(* IEC 61131-3 sources: SmartHomeNew/snapshots/2026-05-25 (part 5) *)

(* ---- PRG_Forensic_Evidence_Governor.st ---- *)
PROGRAM PRG_Forensic_Evidence_Governor
VAR
    L_Now_MS : UDINT;
    L_Forensic_Valid : BOOL := TRUE;
    L_Error_Code : UDINT := 0;
    L_Error_Text : STRING(160) := '';
END_VAR

L_Now_MS := GVL_STATUS.G_System_Time_MS;
L_Forensic_Valid := TRUE;
L_Error_Code := 0;
L_Error_Text := '';

// Fail-safe defaults.
GVL_FORENSIC_EVIDENCE_FABRIC.Forensic_Evidence_Valid := FALSE;
GVL_FORENSIC_EVIDENCE_FABRIC.Forensic_Evidence_Granted := FALSE;
GVL_FORENSIC_EVIDENCE_FABRIC.Forensic_Evidence_Quarantine_Active := TRUE;

GVL_FORENSIC_EVIDENCE_FABRIC.Authority_Lineage_Reconstructable := FALSE;
GVL_FORENSIC_EVIDENCE_FABRIC.Decision_Causality_Traceable := FALSE;
GVL_FORENSIC_EVIDENCE_FABRIC.Distributed_Evidence_Coherent := FALSE;
GVL_FORENSIC_EVIDENCE_FABRIC.Immutable_Audit_Continuity_Valid := FALSE;
GVL_FORENSIC_EVIDENCE_FABRIC.Recovery_Lineage_Preserved := FALSE;

// Compliance federation required.
IF NOT GVL_COMPLIANCE_FEDERATION_FABRIC.Compliance_Federation_Granted THEN
    L_Forensic_Valid := FALSE;
    L_Error_Code := 43000;
    L_Error_Text := 'Compliance federation authority not granted';
END_IF;

// Forensic split-brain detectors.
IF GVL_FORENSIC_EVIDENCE_FABRIC.Authority_Lineage_Gap_Detected THEN
    L_Forensic_Valid := FALSE;
    L_Error_Code := 43001;
    L_Error_Text := 'Authority lineage gap detected';
END_IF;

IF GVL_FORENSIC_EVIDENCE_FABRIC.NonReconstructable_Decision_Detected THEN
    L_Forensic_Valid := FALSE;
    L_Error_Code := 43002;
    L_Error_Text := 'Non-reconstructable decision detected';
END_IF;

IF GVL_FORENSIC_EVIDENCE_FABRIC.History_Evidence_Divergence_Detected THEN
    L_Forensic_Valid := FALSE;
    L_Error_Code := 43003;
    L_Error_Text := 'History evidence divergence detected';
END_IF;

IF GVL_FORENSIC_EVIDENCE_FABRIC.Causal_Chain_Erosion_Detected THEN
    L_Forensic_Valid := FALSE;
    L_Error_Code := 43004;
    L_Error_Text := 'Causal chain erosion detected';
END_IF;

IF GVL_FORENSIC_EVIDENCE_FABRIC.Distributed_Forensic_Inconsistency_Detected THEN
    L_Forensic_Valid := FALSE;
    L_Error_Code := 43005;
    L_Error_Text := 'Distributed forensic inconsistency detected';
END_IF;

IF GVL_FORENSIC_EVIDENCE_FABRIC.Immutable_Audit_Discontinuity_Detected THEN
    L_Forensic_Valid := FALSE;
    L_Error_Code := 43006;
    L_Error_Text := 'Immutable audit discontinuity detected';
END_IF;

// Forensic reconstruction validation.
IF L_Forensic_Valid
AND NOT GVL_FORENSIC_EVIDENCE_FABRIC.Historical_Proof_Chain_Valid THEN
    L_Forensic_Valid := FALSE;
    L_Error_Code := 43010;
    L_Error_Text := 'Historical proof chain invalid';
END_IF;

IF L_Forensic_Valid
AND NOT GVL_FORENSIC_EVIDENCE_FABRIC.Governance_Event_Lineage_Coherent THEN
    L_Forensic_Valid := FALSE;
    L_Error_Code := 43011;
    L_Error_Text := 'Governance event lineage coherence invalid';
END_IF;

IF L_Forensic_Valid
AND NOT GVL_FORENSIC_EVIDENCE_FABRIC.Semantic_Transition_Traceable THEN
    L_Forensic_Valid := FALSE;
    L_Error_Code := 43012;
    L_Error_Text := 'Semantic transition traceability invalid';
END_IF;

IF L_Forensic_Valid
AND NOT GVL_FORENSIC_EVIDENCE_FABRIC.Physical_Transition_Traceable THEN
    L_Forensic_Valid := FALSE;
    L_Error_Code := 43013;
    L_Error_Text := 'Physical transition traceability invalid';
END_IF;

IF L_Forensic_Valid THEN
    GVL_FORENSIC_EVIDENCE_FABRIC.Forensic_Evidence_Valid := TRUE;
    GVL_FORENSIC_EVIDENCE_FABRIC.Forensic_Evidence_Granted := TRUE;
    GVL_FORENSIC_EVIDENCE_FABRIC.Forensic_Evidence_Quarantine_Active := FALSE;

    GVL_FORENSIC_EVIDENCE_FABRIC.Authority_Lineage_Reconstructable := TRUE;
    GVL_FORENSIC_EVIDENCE_FABRIC.Decision_Causality_Traceable := TRUE;
    GVL_FORENSIC_EVIDENCE_FABRIC.Distributed_Evidence_Coherent := TRUE;
    GVL_FORENSIC_EVIDENCE_FABRIC.Immutable_Audit_Continuity_Valid := TRUE;
    GVL_FORENSIC_EVIDENCE_FABRIC.Recovery_Lineage_Preserved := TRUE;

    GVL_FORENSIC_EVIDENCE_FABRIC.Forensic_Evidence_Epoch :=
        GVL_COMPLIANCE_FEDERATION_FABRIC.Compliance_Federation_Epoch;

    GVL_FORENSIC_EVIDENCE_FABRIC.Forensic_Evidence_Epoch_Coherent := TRUE;

    GVL_FORENSIC_EVIDENCE_FABRIC.Forensic_Evidence_Last_Update_MS :=
        L_Now_MS;

    GVL_FORENSIC_EVIDENCE_FABRIC.Forensic_Evidence_Lease_Expired := FALSE;

    GVL_FORENSIC_EVIDENCE_FABRIC.Forensic_Evidence_Last_Error_Code := 0;
    GVL_FORENSIC_EVIDENCE_FABRIC.Forensic_Evidence_Last_Error_Text := '';
ELSE
    GVL_FORENSIC_EVIDENCE_FABRIC.Forensic_Evidence_Valid := FALSE;
    GVL_FORENSIC_EVIDENCE_FABRIC.Forensic_Evidence_Granted := FALSE;
    GVL_FORENSIC_EVIDENCE_FABRIC.Forensic_Evidence_Quarantine_Active := TRUE;

    GVL_FORENSIC_EVIDENCE_FABRIC.Forensic_Evidence_Lease_Expired := TRUE;

    GVL_FORENSIC_EVIDENCE_FABRIC.Forensic_Evidence_Last_Error_Code :=
        L_Error_Code;

    GVL_FORENSIC_EVIDENCE_FABRIC.Forensic_Evidence_Last_Error_Text :=
        L_Error_Text;

    GVL_FORENSIC_EVIDENCE_FABRIC.Forensic_Evidence_Invalidation_Count :=
        GVL_FORENSIC_EVIDENCE_FABRIC.Forensic_Evidence_Invalidation_Count + 1;
END_IF;

END_PROGRAM

(* ---- PRG_Governance_Liveness_Integrity_Governor.st ---- *)
PROGRAM PRG_Governance_Liveness_Integrity_Governor
VAR
    L_Now_MS : UDINT;
    L_Integrity_Valid : BOOL := TRUE;
    L_Error_Code : UDINT := 0;
    L_Error_Text : STRING(160) := '';
END_VAR

L_Now_MS := GVL_STATUS.G_System_Time_MS;
L_Integrity_Valid := TRUE;
L_Error_Code := 0;
L_Error_Text := '';

// Fail-safe defaults.
GVL_GOVERNANCE_LIVENESS_INTEGRITY_FABRIC.Governance_Liveness_Integrity_Valid := FALSE;
GVL_GOVERNANCE_LIVENESS_INTEGRITY_FABRIC.Governance_Liveness_Integrity_Granted := FALSE;
GVL_GOVERNANCE_LIVENESS_INTEGRITY_FABRIC.Governance_Liveness_Integrity_Quarantine_Active := TRUE;

GVL_GOVERNANCE_LIVENESS_INTEGRITY_FABRIC.Governance_Execution_Liveness_Stable := FALSE;
GVL_GOVERNANCE_LIVENESS_INTEGRITY_FABRIC.Integrity_Governor_Scheduling_Canonical := FALSE;
GVL_GOVERNANCE_LIVENESS_INTEGRITY_FABRIC.CrossGovernor_Execution_Continuity_Valid := FALSE;
GVL_GOVERNANCE_LIVENESS_INTEGRITY_FABRIC.Deterministic_Validation_Cycle_Integrity := FALSE;
GVL_GOVERNANCE_LIVENESS_INTEGRITY_FABRIC.Governance_Runtime_Liveness_Coherent := FALSE;

// Governance validator integrity required.
IF NOT GVL_GOVERNANCE_VALIDATOR_INTEGRITY_FABRIC.Governance_Validator_Integrity_Granted THEN
    L_Integrity_Valid := FALSE;
    L_Error_Code := 54000;
    L_Error_Text := 'Governance validator integrity not granted';
END_IF;

// Governance liveness degradation detectors.
IF GVL_GOVERNANCE_LIVENESS_INTEGRITY_FABRIC.Integrity_Governor_Starvation_Detected THEN
    L_Integrity_Valid := FALSE;
    L_Error_Code := 54001;
    L_Error_Text := 'Integrity governor starvation detected';
END_IF;

IF GVL_GOVERNANCE_LIVENESS_INTEGRITY_FABRIC.Validation_Cycle_Skip_Detected THEN
    L_Integrity_Valid := FALSE;
    L_Error_Code := 54002;
    L_Error_Text := 'Validation cycle skip detected';
END_IF;

IF GVL_GOVERNANCE_LIVENESS_INTEGRITY_FABRIC.CrossGovernor_Execution_Jitter_Fork THEN
    L_Integrity_Valid := FALSE;
    L_Error_Code := 54003;
    L_Error_Text := 'Cross-governor execution jitter fork detected';
END_IF;

IF GVL_GOVERNANCE_LIVENESS_INTEGRITY_FABRIC.Selective_Governance_Degradation_Detected THEN
    L_Integrity_Valid := FALSE;
    L_Error_Code := 54004;
    L_Error_Text := 'Selective governance degradation detected';
END_IF;

IF GVL_GOVERNANCE_LIVENESS_INTEGRITY_FABRIC.Runtime_Governor_Execution_Stall_Detected THEN
    L_Integrity_Valid := FALSE;
    L_Error_Code := 54005;
    L_Error_Text := 'Runtime governor execution stall detected';
END_IF;

IF GVL_GOVERNANCE_LIVENESS_INTEGRITY_FABRIC.Distributed_Liveness_Reality_Fork_Detected THEN
    L_Integrity_Valid := FALSE;
    L_Error_Code := 54006;
    L_Error_Text := 'Distributed liveness reality fork detected';
END_IF;

// Governance liveness validation.
IF L_Integrity_Valid
AND NOT GVL_GOVERNANCE_LIVENESS_INTEGRITY_FABRIC.Validation_Cycle_Timing_Monotonic THEN
    L_Integrity_Valid := FALSE;
    L_Error_Code := 54010;
    L_Error_Text := 'Validation cycle timing invalid';
END_IF;

IF L_Integrity_Valid
AND NOT GVL_GOVERNANCE_LIVENESS_INTEGRITY_FABRIC.Distributed_Governor_Execution_Aligned THEN
    L_Integrity_Valid := FALSE;
    L_Error_Code := 54011;
    L_Error_Text := 'Distributed governor execution alignment invalid';
END_IF;

IF L_Integrity_Valid
AND NOT GVL_GOVERNANCE_LIVENESS_INTEGRITY_FABRIC.Runtime_Integrity_Causality_Grounded THEN
    L_Integrity_Valid := FALSE;
    L_Error_Code := 54012;
    L_Error_Text := 'Runtime integrity causality invalid';
END_IF;

IF L_Integrity_Valid
AND NOT GVL_GOVERNANCE_LIVENESS_INTEGRITY_FABRIC.Governance_Execution_Budget_Stable THEN
    L_Integrity_Valid := FALSE;
    L_Error_Code := 54013;
    L_Error_Text := 'Governance execution budget invalid';
END_IF;

IF L_Integrity_Valid THEN
    GVL_GOVERNANCE_LIVENESS_INTEGRITY_FABRIC.Governance_Liveness_Integrity_Valid := TRUE;
    GVL_GOVERNANCE_LIVENESS_INTEGRITY_FABRIC.Governance_Liveness_Integrity_Granted := TRUE;
    GVL_GOVERNANCE_LIVENESS_INTEGRITY_FABRIC.Governance_Liveness_Integrity_Quarantine_Active := FALSE;

    GVL_GOVERNANCE_LIVENESS_INTEGRITY_FABRIC.Governance_Execution_Liveness_Stable := TRUE;
    GVL_GOVERNANCE_LIVENESS_INTEGRITY_FABRIC.Integrity_Governor_Scheduling_Canonical := TRUE;
    GVL_GOVERNANCE_LIVENESS_INTEGRITY_FABRIC.CrossGovernor_Execution_Continuity_Valid := TRUE;
    GVL_GOVERNANCE_LIVENESS_INTEGRITY_FABRIC.Deterministic_Validation_Cycle_Integrity := TRUE;
    GVL_GOVERNANCE_LIVENESS_INTEGRITY_FABRIC.Governance_Runtime_Liveness_Coherent := TRUE;

    GVL_GOVERNANCE_LIVENESS_INTEGRITY_FABRIC.Governance_Liveness_Integrity_Epoch :=
        GVL_GOVERNANCE_VALIDATOR_INTEGRITY_FABRIC.Governance_Validator_Integrity_Epoch;

    GVL_GOVERNANCE_LIVENESS_INTEGRITY_FABRIC.Governance_Liveness_Integrity_Epoch_Coherent := TRUE;

    GVL_GOVERNANCE_LIVENESS_INTEGRITY_FABRIC.Governance_Liveness_Integrity_Last_Update_MS :=
        L_Now_MS;

    GVL_GOVERNANCE_LIVENESS_INTEGRITY_FABRIC.Governance_Liveness_Integrity_Lease_Expired := FALSE;

    GVL_GOVERNANCE_LIVENESS_INTEGRITY_FABRIC.Governance_Liveness_Integrity_Last_Error_Code := 0;
    GVL_GOVERNANCE_LIVENESS_INTEGRITY_FABRIC.Governance_Liveness_Integrity_Last_Error_Text := '';
ELSE
    GVL_GOVERNANCE_LIVENESS_INTEGRITY_FABRIC.Governance_Liveness_Integrity_Valid := FALSE;
    GVL_GOVERNANCE_LIVENESS_INTEGRITY_FABRIC.Governance_Liveness_Integrity_Granted := FALSE;
    GVL_GOVERNANCE_LIVENESS_INTEGRITY_FABRIC.Governance_Liveness_Integrity_Quarantine_Active := TRUE;

    GVL_GOVERNANCE_LIVENESS_INTEGRITY_FABRIC.Governance_Liveness_Integrity_Lease_Expired := TRUE;

    GVL_GOVERNANCE_LIVENESS_INTEGRITY_FABRIC.Governance_Liveness_Integrity_Last_Error_Code :=
        L_Error_Code;

    GVL_GOVERNANCE_LIVENESS_INTEGRITY_FABRIC.Governance_Liveness_Integrity_Last_Error_Text :=
        L_Error_Text;

    GVL_GOVERNANCE_LIVENESS_INTEGRITY_FABRIC.Governance_Liveness_Integrity_Invalidation_Count :=
        GVL_GOVERNANCE_LIVENESS_INTEGRITY_FABRIC.Governance_Liveness_Integrity_Invalidation_Count + 1;
END_IF;

END_PROGRAM

(* ---- PRG_HA_Session_Replication.st ---- *)
PROGRAM PRG_HA_Session_Replication
// ======================================================
// HA SESSION REPLICATION
// ======================================================
// Dedicated HA/session replication boundary.
//
// Purpose:
// replicate canonical peer-session state through isolated
// HA replication surface.
//
// Current implementation:
// bounded loopback foundation.
//
// Future implementations may replace this with:
// - SysCom HA channel
// - shared-memory replication
// - dedicated Ethernet HA link
// - deterministic fieldbus synchronization
//
// without changing distributed governors.
// ======================================================

IF NOT GVL_HA_SESSION_REPLICATION.HA_Replication_Enabled THEN
    GVL_HA_SESSION_REPLICATION.HA_Channel_Healthy := FALSE;
    RETURN;
END_IF;

// ------------------------------------------------------
// Canonical session export replication.
// ------------------------------------------------------

GVL_HA_SESSION_REPLICATION.HA_Remote_Session_Valid :=
    GVL_PEER_SESSION.Remote_Session_Valid;

GVL_HA_SESSION_REPLICATION.HA_Remote_Last_Refresh_MS :=
    GVL_PEER_SESSION.Remote_Last_Refresh_MS;

GVL_HA_SESSION_REPLICATION.HA_Remote_Runtime_Epoch :=
    GVL_PEER_SESSION.Remote_Runtime_Epoch;

GVL_HA_SESSION_REPLICATION.HA_Remote_Snapshot_Epoch :=
    GVL_PEER_SESSION.Remote_Snapshot_Epoch;

GVL_HA_SESSION_REPLICATION.HA_Remote_Boot_Generation :=
    GVL_PEER_SESSION.Remote_Boot_Generation;

GVL_HA_SESSION_REPLICATION.HA_Remote_Fencing_Token :=
    GVL_PEER_SESSION.Remote_Fencing_Token;

GVL_HA_SESSION_REPLICATION.HA_Remote_Publication_Allowed :=
    GVL_PEER_SESSION.Remote_Publication_Allowed;

GVL_HA_SESSION_REPLICATION.HA_Remote_Runtime_Healthy :=
    GVL_PEER_SESSION.Remote_Runtime_Healthy;

GVL_HA_SESSION_REPLICATION.HA_Last_TX_MS :=
    GVL_STATUS.G_System_Time_MS;

GVL_HA_SESSION_REPLICATION.HA_Last_RX_MS :=
    GVL_STATUS.G_System_Time_MS;

GVL_HA_SESSION_REPLICATION.HA_Channel_Healthy := TRUE;

// >>> BULK_SYNC_ANCHOR: PRG_HA_Session_Replication <<<
END_PROGRAM

(* ---- PRG_Heating_Config_Defaults.st ---- *)
PROGRAM PRG_Heating_Config_Defaults
VAR
    L_i : INT;
    L_Manifold : BYTE;
END_VAR

// Default per-circuit comfort/economy profiles.
// This initializer only fills empty records and does not overwrite HMI-edited
// records after circuit_id has been assigned.
FOR L_i := 1 TO GVL_CONSTANTS.C_MAX_HEATING_CIRCUITS DO
    IF GVL_CONFIG.G_HMI_FloorHeating_Configs[L_i].circuit_id = 0 THEN
        CASE L_i OF
            1, 2, 3, 4:
                L_Manifold := 1;
            5, 6, 7, 8:
                L_Manifold := 2;
            9, 10, 11, 12:
                L_Manifold := 3;
            13, 14:
                L_Manifold := 4;
        ELSE
                L_Manifold := 5;
        END_CASE;

        GVL_CONFIG.G_HMI_FloorHeating_Configs[L_i].circuit_id := TO_BYTE(L_i);
        GVL_CONFIG.G_HMI_FloorHeating_Configs[L_i].zone := TO_BYTE(L_i);
        GVL_CONFIG.G_HMI_FloorHeating_Configs[L_i].manifold_id := L_Manifold;
        GVL_CONFIG.G_HMI_FloorHeating_Configs[L_i].sensor_id := TO_BYTE(L_i);
        GVL_CONFIG.G_HMI_FloorHeating_Configs[L_i].valve_id := TO_BYTE(L_i);
        GVL_CONFIG.G_HMI_FloorHeating_Configs[L_i].control_type := 1;

        // Historical design_temp is kept, but explicit comfort_temp is now the
        // room comfort setpoint used by FB_Heating_Circuit_Control.
        GVL_CONFIG.G_HMI_FloorHeating_Configs[L_i].design_temp := 22.0;
        GVL_CONFIG.G_HMI_FloorHeating_Configs[L_i].use_in_normal := TRUE;
        GVL_CONFIG.G_HMI_FloorHeating_Configs[L_i].use_in_away_preheat := TRUE;
        GVL_CONFIG.G_HMI_FloorHeating_Configs[L_i].comfort_temp := 22.0;
        GVL_CONFIG.G_HMI_FloorHeating_Configs[L_i].economy_temp := 17.0;
        GVL_CONFIG.G_HMI_FloorHeating_Configs[L_i].long_away_temp := 12.0;

        GVL_CONFIG.G_HMI_FloorHeating_Configs[L_i].min_temp := 5.0;
        GVL_CONFIG.G_HMI_FloorHeating_Configs[L_i].max_temp := 30.0;
        GVL_CONFIG.G_HMI_FloorHeating_Configs[L_i].pid_kp := 2.0;
        GVL_CONFIG.G_HMI_FloorHeating_Configs[L_i].pwm_period_s := 600;
    END_IF;
END_FOR;

PRG_Away_Heating_HMI_Applicator();

END_PROGRAM

(* ---- PRG_Industrial_Maintainability_Governor.st ---- *)
PROGRAM PRG_Industrial_Maintainability_Governor

// Passive maintainability governance placeholder.
// Runtime maintainability state is currently represented by fabric GVLs only.
// This program is intentionally side-effect free until ownership is formalized.

END_PROGRAM

(* ---- PRG_Input_Quality_Read.st ---- *)
PROGRAM PRG_Input_Quality_Read
VAR
    L_i : INT;
    fbRoomTempQuality : ARRAY[1..GVL_CONSTANTS.C_MAX_ZONES] OF FB_Input_Quality_Observer;
    fbFloorTempQuality : ARRAY[1..GVL_CONSTANTS.C_MAX_HEATING_CIRCUITS] OF FB_Input_Quality_Observer;
END_VAR

FOR L_i := 1 TO GVL_CONSTANTS.C_MAX_ZONES DO
    fbRoomTempQuality[L_i](
        VI_Enable := GVL_INPUT_VALIDATION_CONFIG.G_Enable_Temporal_Anomaly_Detection,
        VI_Value := GVL_STATE.G_Room_Temps[L_i],
        VI_System_Time_MS := GVL_STATUS.G_System_Time_MS,
        VI_Spike_Threshold := GVL_INPUT_VALIDATION_CONFIG.G_Room_Temp_Spike_Threshold,
        VI_Stuck_Timeout_MS := GVL_INPUT_VALIDATION_CONFIG.G_Sensor_Stuck_Timeout_MS,
        VO_Quality => GVL_INPUT_QUALITY.G_Room_Temp_Quality[L_i]
    );
END_FOR;

FOR L_i := 1 TO GVL_CONSTANTS.C_MAX_HEATING_CIRCUITS DO
    fbFloorTempQuality[L_i](
        VI_Enable := GVL_INPUT_VALIDATION_CONFIG.G_Enable_Temporal_Anomaly_Detection,
        VI_Value := GVL_STATE.G_Floor_Temps[L_i],
        VI_System_Time_MS := GVL_STATUS.G_System_Time_MS,
        VI_Spike_Threshold := GVL_INPUT_VALIDATION_CONFIG.G_Room_Temp_Spike_Threshold,
        VI_Stuck_Timeout_MS := GVL_INPUT_VALIDATION_CONFIG.G_Sensor_Stuck_Timeout_MS,
        VO_Quality => GVL_INPUT_QUALITY.G_Floor_Temp_Quality[L_i]
    );
END_FOR;

END_PROGRAM

(* ---- PRG_IO_Read_Discrete_03_Safety_Sensors.st ---- *)
PROGRAM PRG_IO_Read_Discrete_03_Safety_Sensors
VAR
    L_i : INT;
    L_Debounce_Time : TIME := T#100MS;

    fbDebounce_Flood : ARRAY[1..GVL_CONSTANTS.C_MAX_FLOOD_SENSORS] OF FB_System_Timer;
    fbDebounce_Smoke : ARRAY[1..GVL_CONSTANTS.C_MAX_SMOKE_SENSORS] OF FB_System_Timer;
END_VAR

FOR L_i := 1 TO GVL_CONSTANTS.C_MAX_FLOOD_SENSORS DO
    fbDebounce_Flood[L_i](
        IN := GVL_IO.DI_Flood_Sensors[L_i],
        PT := L_Debounce_Time,
        VI_System_Time_MS := GVL_STATUS.G_System_Time_MS
    );
    GVL_STATE.G_Water_Sensors[L_i] := fbDebounce_Flood[L_i].Q;
END_FOR;

FOR L_i := 1 TO GVL_CONSTANTS.C_MAX_SMOKE_SENSORS DO
    fbDebounce_Smoke[L_i](
        IN := GVL_IO.DI_Smoke_Sensors[L_i],
        PT := L_Debounce_Time,
        VI_System_Time_MS := GVL_STATUS.G_System_Time_MS
    );
    GVL_STATE.G_Smoke_Sensors[L_i] := fbDebounce_Smoke[L_i].Q;
END_FOR;

// >>> BULK_SYNC_ANCHOR: PRG_IO_Read_Discrete_03_Safety_Sensors <<<
END_PROGRAM

(* ---- PRG_IO_Read_Manifold_01_Pressure_Current.st ---- *)
PROGRAM PRG_IO_Read_Manifold_01_Pressure_Current
VAR
    L_i : INT;
    L_Manifold_Pressure_Raw : WORD;
    L_Manifold_Current_Raw : WORD;

    fbDiagEventManager : FB_Diagnostics_Event_Manager;
    fbAnalog_Manifold_Pressure : ARRAY[1..GVL_CONSTANTS.C_MAX_MANIFOLDS] OF FB_Sensor_Analog_Processing;
    fbAnalog_Manifold_Current : ARRAY[1..GVL_CONSTANTS.C_MAX_MANIFOLDS] OF FB_Sensor_Analog_Processing;
END_VAR

GVL_STATUS.G_Diagnostics.Manifold_Pressure_Fault_Active := FALSE;
GVL_STATUS.G_Diagnostics.Manifold_Pressure_First_Fault_Index := 0;
GVL_STATUS.G_Diagnostics.Manifold_Current_Fault_Active := FALSE;
GVL_STATUS.G_Diagnostics.Manifold_Current_First_Fault_Index := 0;
GVL_STATUS.G_Diagnostics.Manifold_Pressure_Fault_Text := '';
GVL_STATUS.G_Diagnostics.Manifold_Current_Fault_Text := '';

FOR L_i := 1 TO GVL_CONSTANTS.C_MAX_MANIFOLDS DO
    IF GVL_IO.AI_Manifold_Pressures[L_i] < 0 THEN
        L_Manifold_Pressure_Raw := 0;
    ELSE
        L_Manifold_Pressure_Raw := INT_TO_WORD(GVL_IO.AI_Manifold_Pressures[L_i]);
    END_IF;

    IF GVL_IO.AI_Manifold_Currents[L_i] < 0 THEN
        L_Manifold_Current_Raw := 0;
    ELSE
        L_Manifold_Current_Raw := INT_TO_WORD(GVL_IO.AI_Manifold_Currents[L_i]);
    END_IF;

    fbAnalog_Manifold_Pressure[L_i](
        VI_Raw_Value := L_Manifold_Pressure_Raw,
        VI_Sensor_Type := 0,
        VI_Min_Scale := 0.0,
        VI_Max_Scale := 10.0,
        VI_Offset := 0.0,
        VI_Multiplier := 1.0,
        VI_Filter_Time_MS := GVL_CONSTANTS.C_MS_IN_SECOND,
        VI_System_Time_MS := GVL_STATUS.G_System_Time_MS,
        VI_Fallback_Mode := 0,
        VI_Default_Value := 0.0
    );
    GVL_STATE.G_Manifold_Pressures[L_i] := fbAnalog_Manifold_Pressure[L_i].VO_Value;
    GVL_STATUS.G_Diagnostics.Manifold_Pressure_Fault[L_i] := fbAnalog_Manifold_Pressure[L_i].VO_Error;
    GVL_STATUS.G_Diagnostics.Manifold_Pressure_Diag_Code[L_i] := fbAnalog_Manifold_Pressure[L_i].VO_Diag_Code;

    fbDiagEventManager(
        VI_Code := GVL_CONFIG.ERR_PRESSURE_OUT_OF_RANGE,
        VI_Severity := 3,
        VI_Active := fbAnalog_Manifold_Pressure[L_i].VO_Error,
        VI_Timestamp := GVL_STATUS.G_System_Time_MS,
        VI_Source := 100 + L_i,
        VIO_Events := GVL_STATUS.G_Diagnostics_Events,
        VIO_Count := GVL_STATUS.G_Diagnostics_Count
    );

    fbAnalog_Manifold_Current[L_i](
        VI_Raw_Value := L_Manifold_Current_Raw,
        VI_Sensor_Type := 0,
        VI_Min_Scale := 0.0,
        VI_Max_Scale := 16.0,
        VI_Offset := 0.0,
        VI_Multiplier := 1.0,
        VI_Filter_Time_MS := GVL_CONSTANTS.C_MS_IN_SECOND,
        VI_System_Time_MS := GVL_STATUS.G_System_Time_MS,
        VI_Fallback_Mode := 0,
        VI_Default_Value := 0.0
    );
    GVL_STATE.G_Manifold_Currents[L_i] := fbAnalog_Manifold_Current[L_i].VO_Value;
    GVL_STATUS.G_Diagnostics.Manifold_Current_Fault[L_i] := fbAnalog_Manifold_Current[L_i].VO_Error;
    GVL_STATUS.G_Diagnostics.Manifold_Current_Diag_Code[L_i] := fbAnalog_Manifold_Current[L_i].VO_Diag_Code;

    fbDiagEventManager(
        VI_Code := GVL_CONFIG.ERR_PUMP_UNDERCURRENT,
        VI_Severity := 3,
        VI_Active := fbAnalog_Manifold_Current[L_i].VO_Error,
        VI_Timestamp := GVL_STATUS.G_System_Time_MS,
        VI_Source := 200 + L_i,
        VIO_Events := GVL_STATUS.G_Diagnostics_Events,
        VIO_Count := GVL_STATUS.G_Diagnostics_Count
    );

    IF GVL_STATUS.G_Diagnostics.Manifold_Pressure_Fault[L_i] OR GVL_STATUS.G_Diagnostics.Manifold_Current_Fault[L_i] THEN
        GVL_STATUS.G_Diagnostics.Sensor_Fault := TRUE;
        GVL_STATUS.G_Diagnostics.Subsystem_Degraded := TRUE;
    END_IF;

    IF GVL_STATUS.G_Diagnostics.Manifold_Pressure_Fault[L_i] AND GVL_STATUS.G_Diagnostics.Manifold_Current_Fault[L_i] THEN
        GVL_STATUS.G_Diagnostics.Manifold_Pressure_Fault_Text := 'Correlated pressure/current fault detected';
        GVL_STATUS.G_Diagnostics.Manifold_Current_Fault_Text := 'Correlated pressure/current fault detected';
    ELSIF GVL_STATUS.G_Diagnostics.Manifold_Pressure_Fault[L_i] AND (GVL_STATUS.G_Diagnostics.Manifold_Pressure_Fault_Text = '') THEN
        GVL_STATUS.G_Diagnostics.Manifold_Pressure_Fault_Text := 'Pressure sensor fault detected';
    ELSIF GVL_STATUS.G_Diagnostics.Manifold_Current_Fault[L_i] AND (GVL_STATUS.G_Diagnostics.Manifold_Current_Fault_Text = '') THEN
        GVL_STATUS.G_Diagnostics.Manifold_Current_Fault_Text := 'Current sensor fault detected';
    END_IF;
END_FOR;

// >>> BULK_SYNC_ANCHOR: PRG_IO_Read_Manifold_01_Pressure_Current <<<
END_PROGRAM

(* ---- PRG_IO_Read_Manifold_02_Temperature_Status.st ---- *)
PROGRAM PRG_IO_Read_Manifold_02_Temperature_Status
VAR
    L_i : INT;

    fbCalib_Manifold_T_Supply : ARRAY[1..GVL_CONSTANTS.C_MAX_MANIFOLDS] OF FB_Sensor_Calibration_Processor;
    fbCalib_Manifold_T_Return : ARRAY[1..GVL_CONSTANTS.C_MAX_MANIFOLDS] OF FB_Sensor_Calibration_Processor;
END_VAR

FOR L_i := 1 TO GVL_CONSTANTS.C_MAX_MANIFOLDS DO
    IF GVL_IO.AI_Manifold_Temps_Supply[L_i].wStatus = 0 THEN
        fbCalib_Manifold_T_Supply[L_i](
            VI_Raw_Value := GVL_IO.AI_Manifold_Temps_Supply[L_i].rValue,
            VI_Record := GVL_CONFIG.G_Calib_Manifold_T_Supply[L_i]
        );
        GVL_STATE.G_Manifold_T_Supply[L_i] := fbCalib_Manifold_T_Supply[L_i].VO_Calibrated_Value;
        IF fbCalib_Manifold_T_Supply[L_i].VO_Record_Fault THEN
            GVL_STATUS.G_Diagnostics.Sensor_Fault := TRUE;
        END_IF;
    ELSE
        GVL_STATUS.G_Diagnostics.Sensor_Fault := TRUE;
    END_IF;

    fbCalib_Manifold_T_Return[L_i](
        VI_Raw_Value := INT_TO_REAL(GVL_IO.AI_Manifold_Temps_Return[L_i]) / 10.0,
        VI_Record := GVL_CONFIG.G_Calib_Manifold_T_Return[L_i]
    );
    GVL_STATE.G_Manifold_T_Return[L_i] := fbCalib_Manifold_T_Return[L_i].VO_Calibrated_Value;
    IF fbCalib_Manifold_T_Return[L_i].VO_Record_Fault THEN
        GVL_STATUS.G_Diagnostics.Sensor_Fault := TRUE;
    END_IF;

    GVL_STATE.G_Manifold_End_Switches[L_i] := GVL_IO.DI_Manifold_End_Switches[L_i];
END_FOR;

// >>> BULK_SYNC_ANCHOR: PRG_IO_Read_Manifold_02_Temperature_Status <<<
END_PROGRAM

(* ---- PRG_IO_Read_Phase_01_Module_Health.st ---- *)
PROGRAM PRG_IO_Read_Phase_01_Module_Health
VAR
    fbIO_Watchdog_1 : FB_IO_Module_Watchdog;
    fbIO_Watchdog_2 : FB_IO_Module_Watchdog;
    fbDiagEventManager : FB_Diagnostics_Event_Manager;
    L_IO_Error_Active : BOOL;
    L_i : INT;
END_VAR

// Default unused module slots to online so domain loops over C_MAX_MODULES
// do not report false faults for modules without watchdog bindings.
FOR L_i := 1 TO GVL_CONSTANTS.C_MAX_MODULES DO
    GVL_STATUS.G_IO_Modules_Online[L_i] := TRUE;
END_FOR;

fbIO_Watchdog_1(
    VI_System_Time_MS := GVL_STATUS.G_System_Time_MS,
    VI_Module_ID := 1,
    VI_Heartbeat_Signal := GVL_IO.DI_Module_1_Heartbeat,
    VI_Timeout_MS := 2000
);

fbIO_Watchdog_2(
    VI_System_Time_MS := GVL_STATUS.G_System_Time_MS,
    VI_Module_ID := 2,
    VI_Heartbeat_Signal := GVL_IO.DI_Module_2_Heartbeat,
    VI_Timeout_MS := 2000
);

GVL_STATUS.G_IO_Modules_Online[1] := fbIO_Watchdog_1.VO_Module_Online;
GVL_STATUS.G_IO_Modules_Online[2] := fbIO_Watchdog_2.VO_Module_Online;

L_IO_Error_Active := fbIO_Watchdog_1.VO_Error_Active OR fbIO_Watchdog_2.VO_Error_Active;

fbDiagEventManager(
    VI_Code := 16#E001,
    VI_Severity := 4,
    VI_Active := NOT fbIO_Watchdog_1.VO_Module_Online,
    VI_Timestamp := GVL_STATUS.G_System_Time_MS,
    VI_Source := 1,
    VIO_Events := GVL_STATUS.G_Diagnostics_Events,
    VIO_Count := GVL_STATUS.G_Diagnostics_Count
);

fbDiagEventManager(
    VI_Code := 16#E002,
    VI_Severity := 4,
    VI_Active := NOT fbIO_Watchdog_2.VO_Module_Online,
    VI_Timestamp := GVL_STATUS.G_System_Time_MS,
    VI_Source := 2,
    VIO_Events := GVL_STATUS.G_Diagnostics_Events,
    VIO_Count := GVL_STATUS.G_Diagnostics_Count
);

// >>> BULK_SYNC_ANCHOR: PRG_IO_Read_Phase_01_Module_Health <<<
END_PROGRAM

(* ---- PRG_IO_Read_Phase_03_Environment_Sensors.st ---- *)
PROGRAM PRG_IO_Read_Phase_03_Environment_Sensors
VAR
    L_i : INT;
    L_Filtered_Room_Temp : REAL;
    L_Filtered_Floor_Temp : REAL;
    L_Ambient_Lux : REAL;
    L_Any_Sensor_Fault : BOOL;

    fbCalib_Outdoor_Temp : FB_Sensor_Calibration_Processor;
    fbCalib_Ambient_Lux : FB_Sensor_Calibration_Processor;
    fbCalib_Supply_Temps : ARRAY[1..GVL_CONSTANTS.C_MAX_SUPPLY_TEMPS] OF FB_Sensor_Calibration_Processor;
    fbCalib_Room_Temps : ARRAY[1..GVL_CONSTANTS.C_MAX_ZONES] OF FB_Sensor_Calibration_Processor;
    fbCalib_Floor_Temps : ARRAY[1..GVL_CONSTANTS.C_MAX_ZONES] OF FB_Sensor_Calibration_Processor;
    fbCalib_Room_Hum : ARRAY[1..GVL_CONSTANTS.C_MAX_ZONES] OF FB_Sensor_Calibration_Processor;
    fbCalib_Room_CO2 : ARRAY[1..GVL_CONSTANTS.C_MAX_ZONES] OF FB_Sensor_Calibration_Processor;
END_VAR

L_Any_Sensor_Fault := FALSE;

fbCalib_Outdoor_Temp(
    VI_Raw_Value := GVL_IO.AI_Temp_Outdoor.rValue,
    VI_Record := GVL_CONFIG.G_Calib_Outdoor_Temp
);
GVL_STATE.G_Outdoor_Temp := fbCalib_Outdoor_Temp.VO_Calibrated_Value;
IF fbCalib_Outdoor_Temp.VO_Record_Fault THEN
    L_Any_Sensor_Fault := TRUE;
END_IF;

IF GVL_CONFIG.G_Entrance_Light_Assist_Use_Lux_Sensor THEN
    IF GVL_IO.AI_Ambient_Lux.wStatus = 0 THEN
        fbCalib_Ambient_Lux(
            VI_Raw_Value := GVL_IO.AI_Ambient_Lux.rValue,
            VI_Record := GVL_CONFIG.G_Calib_Ambient_Lux
        );
        L_Ambient_Lux := fbCalib_Ambient_Lux.VO_Calibrated_Value;
        IF fbCalib_Ambient_Lux.VO_Record_Fault THEN
            L_Any_Sensor_Fault := TRUE;
        END_IF;

        IF (L_Ambient_Lux < 0.0) OR (L_Ambient_Lux > 200000.0) THEN
            GVL_STATE.G_Ambient_Lux_Sensor_Fault := TRUE;
            GVL_STATE.G_Ambient_Lux_Valid := FALSE;
            L_Any_Sensor_Fault := TRUE;
        ELSE
            GVL_STATE.G_Ambient_Lux := L_Ambient_Lux;
            GVL_STATE.G_Ambient_Lux_Valid := TRUE;
            GVL_STATE.G_Ambient_Lux_Sensor_Fault := FALSE;
        END_IF;
    ELSE
        GVL_STATE.G_Ambient_Lux_Valid := FALSE;
        GVL_STATE.G_Ambient_Lux_Sensor_Fault := TRUE;
        L_Any_Sensor_Fault := TRUE;
    END_IF;
ELSE
    GVL_STATE.G_Ambient_Lux_Valid := FALSE;
    GVL_STATE.G_Ambient_Lux_Sensor_Fault := FALSE;
END_IF;

FOR L_i := 1 TO GVL_CONSTANTS.C_MAX_SUPPLY_TEMPS DO
    IF GVL_IO.AI_Supply_Temps[L_i].wStatus = 0 THEN
        fbCalib_Supply_Temps[L_i](
            VI_Raw_Value := GVL_IO.AI_Supply_Temps[L_i].rValue,
            VI_Record := GVL_CONFIG.G_Calib_Supply_Temps[L_i]
        );
        GVL_STATE.G_Supply_Temps[L_i] := fbCalib_Supply_Temps[L_i].VO_Calibrated_Value;
        IF fbCalib_Supply_Temps[L_i].VO_Record_Fault THEN
            L_Any_Sensor_Fault := TRUE;
        END_IF;
    ELSE
        L_Any_Sensor_Fault := TRUE;
    END_IF;
END_FOR;

FOR L_i := 1 TO GVL_CONSTANTS.C_MAX_ZONES DO
    fbCalib_Room_Hum[L_i](
        VI_Raw_Value := GVL_IO.AI_Room_Hum[L_i],
        VI_Record := GVL_CONFIG.G_Calib_Humidity[L_i]
    );
    GVL_STATE.G_Room_Hum[L_i] := fbCalib_Room_Hum[L_i].VO_Calibrated_Value;
    IF fbCalib_Room_Hum[L_i].VO_Record_Fault THEN
        L_Any_Sensor_Fault := TRUE;
    END_IF;

    fbCalib_Room_CO2[L_i](
        VI_Raw_Value := GVL_IO.AI_Room_CO2[L_i],
        VI_Record := GVL_CONFIG.G_Calib_CO2[L_i]
    );
    GVL_STATE.G_Room_CO2[L_i] := fbCalib_Room_CO2[L_i].VO_Calibrated_Value;
    IF fbCalib_Room_CO2[L_i].VO_Record_Fault THEN
        L_Any_Sensor_Fault := TRUE;
    END_IF;
END_FOR;

FOR L_i := 1 TO GVL_CONSTANTS.C_MAX_ZONES DO
    fbCalib_Room_Temps[L_i](
        VI_Raw_Value := GVL_IO.AI_Room_Temps[L_i],
        VI_Record := GVL_CONFIG.G_Calib_Room_Temps[L_i]
    );
    IF fbCalib_Room_Temps[L_i].VO_Record_Fault THEN
        L_Any_Sensor_Fault := TRUE;
    END_IF;

    IF GVL_STATE.G_Last_Valid_Room_Temps[L_i] = 0.0 THEN
        L_Filtered_Room_Temp := fbCalib_Room_Temps[L_i].VO_Calibrated_Value;
    ELSE
        L_Filtered_Room_Temp := (GVL_STATE.G_Last_Valid_Room_Temps[L_i] * 0.9) + (fbCalib_Room_Temps[L_i].VO_Calibrated_Value * 0.1);
    END_IF;

    IF (L_Filtered_Room_Temp < -50.0) OR (L_Filtered_Room_Temp > 100.0) THEN
        GVL_STATE.G_Temp_Sensor_Fault[L_i] := TRUE;
        GVL_STATE.G_Room_Temps[L_i] := GVL_STATE.G_Last_Valid_Room_Temps[L_i];
        L_Any_Sensor_Fault := TRUE;
    ELSE
        GVL_STATE.G_Temp_Sensor_Fault[L_i] := FALSE;
        GVL_STATE.G_Room_Temps[L_i] := L_Filtered_Room_Temp;
        GVL_STATE.G_Last_Valid_Room_Temps[L_i] := L_Filtered_Room_Temp;
    END_IF;
END_FOR;

FOR L_i := 1 TO GVL_CONSTANTS.C_MAX_HEATING_CIRCUITS DO
    IF L_i <= GVL_CONSTANTS.C_MAX_ZONES THEN
        fbCalib_Floor_Temps[L_i](
            VI_Raw_Value := GVL_IO.AI_Floor_Temps[L_i],
            VI_Record := GVL_CONFIG.G_Calib_Floor_Temps[L_i]
        );
        IF fbCalib_Floor_Temps[L_i].VO_Record_Fault THEN
            L_Any_Sensor_Fault := TRUE;
        END_IF;

        IF GVL_STATE.G_Last_Valid_Floor_Temps[L_i] = 0.0 THEN
            L_Filtered_Floor_Temp := fbCalib_Floor_Temps[L_i].VO_Calibrated_Value;
        ELSE
            L_Filtered_Floor_Temp := (GVL_STATE.G_Last_Valid_Floor_Temps[L_i] * 0.9) + (fbCalib_Floor_Temps[L_i].VO_Calibrated_Value * 0.1);
        END_IF;

        IF (L_Filtered_Floor_Temp < -50.0) OR (L_Filtered_Floor_Temp > 100.0) THEN
            GVL_STATE.G_Floor_Temp_Sensor_Fault[L_i] := TRUE;
            GVL_STATE.G_Floor_Temps[L_i] := GVL_STATE.G_Last_Valid_Floor_Temps[L_i];
            L_Any_Sensor_Fault := TRUE;
        ELSE
            GVL_STATE.G_Floor_Temp_Sensor_Fault[L_i] := FALSE;
            GVL_STATE.G_Floor_Temps[L_i] := L_Filtered_Floor_Temp;
            GVL_STATE.G_Last_Valid_Floor_Temps[L_i] := L_Filtered_Floor_Temp;
        END_IF;
    ELSE
        GVL_STATE.G_Floor_Temp_Sensor_Fault[L_i] := TRUE;
        GVL_STATE.G_Floor_Temps[L_i] := GVL_STATE.G_Last_Valid_Floor_Temps[L_i];
        L_Any_Sensor_Fault := TRUE;
    END_IF;
END_FOR;

GVL_STATUS.G_Diagnostics.Sensor_Fault := L_Any_Sensor_Fault;

// >>> BULK_SYNC_ANCHOR: PRG_IO_Read_Phase_03_Environment_Sensors <<<
END_PROGRAM

(* ---- PRG_IO_Read_Phase_04_Heating_Manifold_Sensors.st ---- *)
PROGRAM PRG_IO_Read_Phase_04_Heating_Manifold_Sensors
// ==============================================================================
// IO READ PHASE 04 — heating manifold analog sensors and status inputs.
// ==============================================================================
// Execution order is preserved from the former phase body.
// No gating, shedding or behavior changes are applied here.
// ==============================================================================

PRG_IO_Read_Manifold_01_Pressure_Current();
PRG_IO_Read_Manifold_02_Temperature_Status();

// >>> BULK_SYNC_ANCHOR: PRG_IO_Read_Phase_04_Heating_Manifold_Sensors <<<
END_PROGRAM

(* ---- PRG_IO_Write.st ---- *)
PROGRAM PRG_IO_Write
// ==============================================================================
// IO WRITE — deterministic physical output publication phase map.
// ==============================================================================
// Execution preserves the former priority model:
// 1. derive publication guards and forced-off flags
// 2. hard-stop safe-state publication and return when required
// 3. normal domain output projection
// 4. final alarm/gas valve and trace publication
// ==============================================================================

PRG_IO_Write_Phase_01_Context();

IF (NOT GVL_STATUS.G_Is_Active_PLC)
   OR GVL_IO_WRITE_RUNTIME_BUFFER.B_Global_Hard_Stop THEN
    PRG_IO_Write_Phase_02_Hard_Stop_Safe_State();
    RETURN;
END_IF;

PRG_IO_Write_Phase_03_Domain_Projection();
PRG_IO_Write_Phase_04_Alarm_Trace();

// >>> BULK_SYNC_ANCHOR: PRG_IO_Write <<<
END_PROGRAM

(* ---- PRG_IO_Write_Phase_03_Domain_Projection.st ---- *)
PROGRAM PRG_IO_Write_Phase_03_Domain_Projection
// IO write phase 03: publish normal domain output projections.
VAR
    L_i : INT;
END_VAR

FOR L_i := 1 TO GVL_CONSTANTS.C_MAX_HEATING_CIRCUITS DO
    IF (L_i > GVL_SYSTEM_SIZE_CONFIG.G_Active_Heating_Circuits)
       OR GVL_IO_WRITE_RUNTIME_BUFFER.B_Heating_Forced_Off THEN
        GVL_IO.DO_Zone_Valves[L_i] := FALSE;
    ELSE
        GVL_IO.DO_Zone_Valves[L_i] := GVL_HEATING_OUTPUT.DO_Zone_Valves[L_i];
    END_IF;
END_FOR;

FOR L_i := 1 TO GVL_CONSTANTS.C_MAX_MANIFOLDS DO
    IF GVL_IO_WRITE_RUNTIME_BUFFER.B_Heating_Forced_Off
       AND NOT (GVL_IO_WRITE_RUNTIME_BUFFER.B_Gas_Safety_Stop
                AND GVL_IO_WRITE_RUNTIME_BUFFER.B_Freeze_Active) THEN
        GVL_IO.DO_Manifold_Pumps[L_i] := FALSE;
        GVL_IO.AO_Manifold_Valves[L_i] := 0;
    ELSE
        GVL_IO.DO_Manifold_Pumps[L_i] := GVL_HEATING_OUTPUT.DO_Manifold_Pumps[L_i];
        GVL_IO.AO_Manifold_Valves[L_i] := GVL_HEATING_OUTPUT.AO_Manifold_Valves[L_i];
    END_IF;
END_FOR;

IF GVL_IO_WRITE_RUNTIME_BUFFER.B_Heating_Forced_Off
   AND NOT (GVL_IO_WRITE_RUNTIME_BUFFER.B_Gas_Safety_Stop
            AND GVL_IO_WRITE_RUNTIME_BUFFER.B_Freeze_Active) THEN
    GVL_IO.DO_DHW_Heating_Pump := FALSE;
    GVL_IO.DO_DHW_Circ_Pump := FALSE;
    GVL_IO.DO_Backup_Circulation_Pump := FALSE;
    GVL_IO.DO_Electric_Heater_Enable := FALSE;
ELSE
    GVL_IO.DO_DHW_Heating_Pump := GVL_HEATING_OUTPUT.DO_DHW_Heating_Pump;
    GVL_IO.DO_DHW_Circ_Pump := GVL_HEATING_OUTPUT.DO_DHW_Circ_Pump;
    GVL_IO.DO_Backup_Circulation_Pump := GVL_HEATING_OUTPUT.DO_Backup_Circulation_Pump;
    GVL_IO.DO_Electric_Heater_Enable := GVL_HEATING_OUTPUT.DO_Electric_Heater_Enable;
END_IF;

FOR L_i := 1 TO GVL_CONSTANTS.C_MAX_SUPPLY_FANS DO
    IF GVL_IO_WRITE_RUNTIME_BUFFER.B_Vent_Forced_Off THEN
        GVL_IO.AO_Supply_Fans[L_i] := 0;
    ELSE
        GVL_IO.AO_Supply_Fans[L_i] := GVL_VENT_OUTPUT.AO_Supply_Fans[L_i];
    END_IF;
END_FOR;

FOR L_i := 1 TO GVL_CONSTANTS.C_MAX_EXHAUST_FANS DO
    IF GVL_IO_WRITE_RUNTIME_BUFFER.B_Vent_Forced_Off THEN
        GVL_IO.AO_Exhaust_Fans[L_i] := 0;
    ELSE
        GVL_IO.AO_Exhaust_Fans[L_i] := GVL_VENT_OUTPUT.AO_Exhaust_Fans[L_i];
    END_IF;
END_FOR;

// Water outputs. PRG_Water owns the domain projection in GVL_WATER_OUTPUT;
// command shadow remains the common-inlet emergency fallback.
IF GVL_IO_WRITE_RUNTIME_BUFFER.B_Water_Forced_Off THEN
    GVL_IO.DO_Water_Valve_35_Open := FALSE;
    GVL_IO.DO_Water_Valve_35_Close := FALSE;
    GVL_IO.DO_Water_Valve_36_Open := FALSE;
    GVL_IO.DO_Water_Valve_36_Close := FALSE;

    FOR L_i := 1 TO 6 DO
        GVL_IO.DO_Water_Local_Valve_Open[L_i] := FALSE;
        GVL_IO.DO_Water_Local_Valve_Close[L_i] := FALSE;
    END_FOR;
ELSE
    GVL_IO.DO_Water_Valve_35_Open := GVL_WATER_OUTPUT.DO_Water_Valve_35_Open;
    GVL_IO.DO_Water_Valve_35_Close := GVL_WATER_OUTPUT.DO_Water_Valve_35_Close OR GVL_COMMAND_SHADOW.G_Close_Valve_35;
    GVL_IO.DO_Water_Valve_36_Open := GVL_WATER_OUTPUT.DO_Water_Valve_36_Open;
    GVL_IO.DO_Water_Valve_36_Close := GVL_WATER_OUTPUT.DO_Water_Valve_36_Close OR GVL_COMMAND_SHADOW.G_Close_Valve_36;

    FOR L_i := 1 TO 6 DO
        GVL_IO.DO_Water_Local_Valve_Open[L_i] := GVL_WATER_OUTPUT.DO_Water_Local_Valve_Open[L_i];
        GVL_IO.DO_Water_Local_Valve_Close[L_i] := GVL_WATER_OUTPUT.DO_Water_Local_Valve_Close[L_i];
    END_FOR;
END_IF;

FOR L_i := 1 TO GVL_CONSTANTS.C_MAX_WATER_ZONES DO
    IF (L_i > GVL_SYSTEM_SIZE_CONFIG.G_Active_Water_Zones)
       OR GVL_IO_WRITE_RUNTIME_BUFFER.B_Water_Forced_Off THEN
        GVL_IO.DO_Water_Zone_Enable[L_i] := FALSE;
    ELSE
        GVL_IO.DO_Water_Zone_Enable[L_i] := GVL_WATER_OUTPUT.DO_Water_Zone_Enable[L_i];
    END_IF;
END_FOR;

FOR L_i := 1 TO GVL_CONSTANTS.C_MAX_LIGHT_ZONES DO
    IF L_i > GVL_SYSTEM_SIZE_CONFIG.G_Active_Light_Zones THEN
        GVL_IO.AO_Lighting_Levels[L_i] := 0;
    ELSE
        GVL_IO.AO_Lighting_Levels[L_i] := GVL_LIGHTING_OUTPUT.AO_Lighting_Levels[L_i];
    END_IF;
END_FOR;

FOR L_i := 1 TO GVL_CONSTANTS.C_MAX_BLINDS DO
    IF L_i > GVL_SYSTEM_SIZE_CONFIG.G_Active_Blinds THEN
        GVL_IO.AO_Blinds_Positions[L_i] := 1000;
    ELSE
        GVL_IO.AO_Blinds_Positions[L_i] := GVL_LIGHTING_OUTPUT.AO_Blinds_Positions[L_i];
    END_IF;
END_FOR;

FOR L_i := 1 TO GVL_CONSTANTS.C_MAX_SOCKETS DO
    IF L_i > GVL_SYSTEM_SIZE_CONFIG.G_Active_Sockets THEN
        GVL_IO.DO_Sockets[L_i] := FALSE;
    ELSE
        GVL_IO.DO_Sockets[L_i] := GVL_LIGHTING_OUTPUT.DO_Sockets[L_i];
    END_IF;
END_FOR;

IF GVL_IO_WRITE_RUNTIME_BUFFER.B_Access_Forced_Off THEN
    GVL_IO.DO_Gate_Open := FALSE;
    GVL_IO.DO_Wicket_Open := FALSE;
    GVL_IO.DO_Lock_1_Open := FALSE;
    GVL_IO.DO_Lock_1_Close := FALSE;
    GVL_IO.DO_Lock_2_Open := FALSE;
    GVL_IO.DO_Lock_2_Close := FALSE;
ELSE
    GVL_IO.DO_Gate_Open := GVL_ACCESS_OUTPUT.DO_Gate_Open;
    GVL_IO.DO_Wicket_Open := GVL_ACCESS_OUTPUT.DO_Wicket_Open;
    GVL_IO.DO_Lock_1_Open := GVL_ACCESS_OUTPUT.DO_Lock_1_Open;
    GVL_IO.DO_Lock_1_Close := GVL_ACCESS_OUTPUT.DO_Lock_1_Close;
    GVL_IO.DO_Lock_2_Open := GVL_ACCESS_OUTPUT.DO_Lock_2_Open;
    GVL_IO.DO_Lock_2_Close := GVL_ACCESS_OUTPUT.DO_Lock_2_Close;
END_IF;

// >>> BULK_SYNC_ANCHOR: PRG_IO_Write_Phase_03_Domain_Projection <<<
END_PROGRAM

(* ---- PRG_Lighting_Phase_01_Context.st ---- *)
PROGRAM PRG_Lighting_Phase_01_Context
VAR
    L_i : INT;
    L_Evac_Blink_Phase : UDINT;
END_VAR

GVL_LIGHTING_RUNTIME_BUFFER.B_Fire_Alarm_Active :=
    GVL_HEALTH_BRIDGE.G_Smoke_Detected
    OR GVL_STATE.G_Safety_Smoke_Latched;

GVL_LIGHTING_RUNTIME_BUFFER.B_Flood_Alarm_Active :=
    GVL_HEALTH_BRIDGE.G_Leak_Detected
    OR GVL_STATE.G_Safety_Leak_Latched;

GVL_LIGHTING_RUNTIME_BUFFER.B_Security_Armed := GVL_ALARM.G_Security_Armed;
GVL_LIGHTING_RUNTIME_BUFFER.B_Security_Alarm := GVL_ALARM.G_Security_Alarm;

L_Evac_Blink_Phase := (GVL_STATUS.G_System_Time_MS / 500) MOD 2;
GVL_LIGHTING_RUNTIME_BUFFER.B_Evac_Blink_On := (L_Evac_Blink_Phase = 0);

GVL_LIGHTING_RUNTIME_BUFFER.B_Distributed_Execute_Allowed :=
    GVL_Distributed_Execution_Gates.G_Can_Execute;

GVL_LIGHTING_RUNTIME_BUFFER.B_Distributed_Projection_Allowed :=
    GVL_Distributed_Execution_Gates.G_Can_Own_Projection;

GVL_LIGHTING_RUNTIME_BUFFER.B_Emergency_Lighting_Override :=
    GVL_STATE.G_Evacuation_Lighting_Active
    OR GVL_LIGHTING_RUNTIME_BUFFER.B_Fire_Alarm_Active;

FOR L_i := 1 TO GVL_CONSTANTS.C_MAX_LIGHT_ZONES DO
    IF GVL_INTENT_SYSTEM.I_Lighting_Overrides_Block OR GVL_SYSTEM_COORDINATION.G_Block_Lighting_Override THEN
        GVL_LIGHTING_RUNTIME_BUFFER.B_Manual_Light_Override[L_i] := 0;
    ELSE
        GVL_LIGHTING_RUNTIME_BUFFER.B_Manual_Light_Override[L_i] := GVL_INTENT_USER.I_Lighting_Override_32[L_i];
    END_IF;

    GVL_LIGHTING_RUNTIME_BUFFER.B_Sim_Lights[L_i] := GVL_STATE.G_Sim_Lights[L_i];
    GVL_LIGHTING_RUNTIME_BUFFER.B_Physical_Switches[L_i] := GVL_STATE.G_Physical_Switches[L_i];
    GVL_LIGHTING_RUNTIME_BUFFER.B_Motion_Sensors[L_i] := GVL_STATE.G_Motion_Sensors[L_i];
END_FOR;

FOR L_i := 1 TO GVL_CONSTANTS.C_MAX_BLINDS DO
    IF GVL_INTENT_SYSTEM.I_Blinds_Overrides_Block THEN
        GVL_LIGHTING_RUNTIME_BUFFER.B_Manual_Blinds_Override[L_i] := 0;
    ELSE
        GVL_LIGHTING_RUNTIME_BUFFER.B_Manual_Blinds_Override[L_i] := GVL_INTENT_USER.I_Blinds_Override_32[L_i];
    END_IF;

    GVL_LIGHTING_RUNTIME_BUFFER.B_Blinds_Override[L_i] :=
        GVL_LIGHTING_RUNTIME_BUFFER.B_Manual_Blinds_Override[L_i];
END_FOR;

FOR L_i := 1 TO GVL_CONSTANTS.C_MAX_SOCKETS DO
    IF GVL_INTENT_SYSTEM.I_Socket_Overrides_Block OR GVL_SYSTEM_COORDINATION.G_Block_Sockets_Override THEN
        GVL_LIGHTING_RUNTIME_BUFFER.B_Manual_Socket_Override[L_i] := FALSE;
    ELSE
        GVL_LIGHTING_RUNTIME_BUFFER.B_Manual_Socket_Override[L_i] := GVL_INTENT_USER.I_Socket_Override_32[L_i];
    END_IF;

    GVL_LIGHTING_RUNTIME_BUFFER.B_Socket_Override[L_i] :=
        GVL_LIGHTING_RUNTIME_BUFFER.B_Manual_Socket_Override[L_i];
END_FOR;

// >>> BULK_SYNC_ANCHOR: PRG_Lighting_Phase_01_Context <<<
END_PROGRAM

(* ---- PRG_Lighting_Phase_03_Priority_Restrictions.st ---- *)
PROGRAM PRG_Lighting_Phase_03_Priority_Restrictions
VAR
    L_i : INT;
END_VAR

// Priority overrides after normal manager calculation:
// Evacuation > Fire > Security Alarm > Security Armed > Normal
IF GVL_STATE.G_Evacuation_Lighting_Active THEN
    FOR L_i := 1 TO GVL_CONSTANTS.C_MAX_LIGHT_ZONES DO
        CASE GVL_STATE.G_Evac_Guidance[L_i] OF
            -1:
                GVL_STATE.G_Lighting_Levels[L_i] := 0;
            1:
                GVL_STATE.G_Lighting_Levels[L_i] := 100;
        ELSE
            IF GVL_LIGHTING_RUNTIME_BUFFER.B_Evac_Blink_On THEN
                GVL_STATE.G_Lighting_Levels[L_i] := 100;
            ELSE
                GVL_STATE.G_Lighting_Levels[L_i] := 0;
            END_IF;
        END_CASE;
    END_FOR;
ELSIF GVL_LIGHTING_RUNTIME_BUFFER.B_Fire_Alarm_Active THEN
    FOR L_i := 1 TO GVL_CONSTANTS.C_MAX_LIGHT_ZONES DO
        GVL_STATE.G_Lighting_Levels[L_i] := 100;
    END_FOR;
    FOR L_i := 1 TO GVL_CONSTANTS.C_MAX_BLINDS DO
        GVL_STATE.G_Blinds_Positions[L_i] := 100;
    END_FOR;
ELSIF GVL_LIGHTING_RUNTIME_BUFFER.B_Security_Alarm THEN
    FOR L_i := 1 TO GVL_CONSTANTS.C_MAX_LIGHT_ZONES DO
        GVL_STATE.G_Lighting_Levels[L_i] := 100;
    END_FOR;
ELSIF GVL_LIGHTING_RUNTIME_BUFFER.B_Security_Armed THEN
    FOR L_i := 1 TO GVL_CONSTANTS.C_MAX_LIGHT_ZONES DO
        GVL_STATE.G_Lighting_Levels[L_i] := 0;
    END_FOR;
END_IF;

// Distributed execution/projection restriction.
// If manager execution or output projection is blocked, clear non-emergency lighting state
// so publication cannot reuse stale values from a previous scan.
IF (
        NOT GVL_LIGHTING_RUNTIME_BUFFER.B_Distributed_Execute_Allowed
        OR NOT GVL_LIGHTING_RUNTIME_BUFFER.B_Distributed_Projection_Allowed
   )
   AND NOT GVL_LIGHTING_RUNTIME_BUFFER.B_Emergency_Lighting_Override THEN

    FOR L_i := 1 TO GVL_CONSTANTS.C_MAX_LIGHT_ZONES DO
        GVL_STATE.G_Lighting_Levels[L_i] := 0;
    END_FOR;

    FOR L_i := 1 TO GVL_CONSTANTS.C_MAX_BLINDS DO
        GVL_STATE.G_Blinds_Positions[L_i] := 100;
    END_FOR;

    FOR L_i := 1 TO GVL_CONSTANTS.C_MAX_SOCKETS DO
        GVL_STATE.G_Socket_States[L_i] := FALSE;
    END_FOR;

END_IF;

// >>> BULK_SYNC_ANCHOR: PRG_Lighting_Phase_03_Priority_Restrictions <<<
END_PROGRAM

(* ---- PRG_Lighting_Phase_04_Output_Publication.st ---- *)
PROGRAM PRG_Lighting_Phase_04_Output_Publication
VAR
    L_i : INT;
    L_Wet_Zone_Any_Active : BOOL;
END_VAR

GVL_LIGHTING_RUNTIME.G_Runtime_Required := FALSE;
GVL_LIGHTING_RUNTIME.G_Runtime_Executed := TRUE;
GVL_LIGHTING_RUNTIME.G_Runtime_Idle_By_Design := FALSE;
GVL_LIGHTING_RUNTIME.G_Runtime_Blocked_By_Distributed_Gates := FALSE;
GVL_LIGHTING_RUNTIME.G_Emergency_Override_Active := GVL_LIGHTING_RUNTIME_BUFFER.B_Emergency_Lighting_Override;
GVL_LIGHTING_RUNTIME.G_Any_Light_Active := FALSE;
GVL_LIGHTING_RUNTIME.G_Any_Blind_Not_Safe_Open := FALSE;
GVL_LIGHTING_RUNTIME.G_Any_Socket_Active := FALSE;
GVL_LIGHTING_RUNTIME.G_Last_Update_MS := GVL_STATUS.G_System_Time_MS;

// Publish wet-zone activity from the final lighting state seen by IO_Write.
L_Wet_Zone_Any_Active := FALSE;
FOR L_i := 1 TO GVL_CONSTANTS.C_MAX_LIGHT_ZONES DO
    IF GVL_CONFIG.G_Wet_Zone_Map[L_i] AND (GVL_STATE.G_Lighting_Levels[L_i] > 10) THEN
        L_Wet_Zone_Any_Active := TRUE;
    END_IF;

    IF GVL_STATE.G_Lighting_Levels[L_i] > 0 THEN
        GVL_LIGHTING_RUNTIME.G_Any_Light_Active := TRUE;
    END_IF;
END_FOR;
GVL_STATUS.G_Wet_Zone_Light_Active := L_Wet_Zone_Any_Active;

// Domain output projection.
FOR L_i := 1 TO GVL_CONSTANTS.C_MAX_LIGHT_ZONES DO
    GVL_LIGHTING_OUTPUT.AO_Lighting_Levels[L_i] := BYTE_TO_UINT(GVL_STATE.G_Lighting_Levels[L_i]) * 10;
END_FOR;

FOR L_i := 1 TO GVL_CONSTANTS.C_MAX_BLINDS DO
    IF GVL_STATE.G_Blinds_Positions[L_i] < 100 THEN
        GVL_LIGHTING_RUNTIME.G_Any_Blind_Not_Safe_Open := TRUE;
    END_IF;

    GVL_LIGHTING_OUTPUT.AO_Blinds_Positions[L_i] := BYTE_TO_UINT(GVL_STATE.G_Blinds_Positions[L_i]) * 10;
END_FOR;

FOR L_i := 1 TO GVL_CONSTANTS.C_MAX_SOCKETS DO
    IF GVL_STATE.G_Socket_States[L_i] THEN
        GVL_LIGHTING_RUNTIME.G_Any_Socket_Active := TRUE;
    END_IF;

    GVL_LIGHTING_OUTPUT.DO_Sockets[L_i] := GVL_STATE.G_Socket_States[L_i];
END_FOR;

GVL_LIGHTING_RUNTIME.G_Runtime_Blocked_By_Distributed_Gates :=
    NOT GVL_LIGHTING_RUNTIME_BUFFER.B_Distributed_Projection_Allowed
    AND NOT GVL_LIGHTING_RUNTIME_BUFFER.B_Emergency_Lighting_Override;

GVL_LIGHTING_RUNTIME.G_Runtime_Required :=
    GVL_LIGHTING_RUNTIME.G_Emergency_Override_Active
    OR GVL_LIGHTING_RUNTIME.G_Any_Light_Active
    OR GVL_LIGHTING_RUNTIME.G_Any_Blind_Not_Safe_Open
    OR GVL_LIGHTING_RUNTIME.G_Any_Socket_Active
    OR GVL_LIGHTING_RUNTIME_BUFFER.B_Security_Armed
    OR GVL_LIGHTING_RUNTIME_BUFFER.B_Security_Alarm;

GVL_LIGHTING_RUNTIME.G_Runtime_Idle_By_Design :=
    NOT GVL_LIGHTING_RUNTIME.G_Runtime_Required;

IF GVL_LIGHTING_RUNTIME.G_Runtime_Blocked_By_Distributed_Gates THEN
    GVL_LIGHTING_RUNTIME.G_Status_Code := 2;
    GVL_LIGHTING_RUNTIME.G_Status_Text := 'Lighting runtime blocked by distributed gates';
ELSIF GVL_LIGHTING_RUNTIME.G_Runtime_Idle_By_Design THEN
    GVL_LIGHTING_RUNTIME.G_Status_Code := 0;
    GVL_LIGHTING_RUNTIME.G_Status_Text := 'Lighting runtime idle by design';
ELSE
    GVL_LIGHTING_RUNTIME.G_Status_Code := 1;
    GVL_LIGHTING_RUNTIME.G_Status_Text := 'Lighting runtime active';
END_IF;

// >>> BULK_SYNC_ANCHOR: PRG_Lighting_Phase_04_Output_Publication <<<
END_PROGRAM

(* ---- PRG_Main_Phase_02_Redundancy.st ---- *)
PROGRAM PRG_Main_Phase_02_Redundancy
// MAIN PHASE 02 — local PLC authority / cold-spare model.
// Critical: yes. Called every PLC scan.
//
// Current architecture: one active PLC controls the system; a second PLC is a
// cold spare only and must not participate in runtime ownership, hot failover,
// direct state replication or physical output arbitration.
VAR
    fbSystemDiagnostics : FB_System_Diagnostics;
    fbServiceHeartbeatTimer : FB_System_Timer;
    L_Service_Heartbeat_State : BOOL;
END_VAR

GVL_MAIN_PHASE_FEEDBACK.G_Current_Phase := 2;

// Local-only authority. No hot standby arbitration is performed in runtime.
GVL_STATUS.G_Is_Active_PLC := TRUE;
GVL_STATUS.G_Other_PLC_Is_Active := FALSE;
GVL_STATUS.G_Remote_PLC_Alive := FALSE;
GVL_STATUS.G_Remote_PLC_Pulse := FALSE;
GVL_STATUS.G_Active_PLC_ID := GVL_STATUS.G_Local_PLC_ID;

// Physical/service status outputs. The heartbeat output is only a local service
// indicator and is not used for automatic failover.
fbServiceHeartbeatTimer(
    IN := NOT fbServiceHeartbeatTimer.Q,
    PT := T#500ms,
    VI_System_Time_MS := GVL_TIME_SERVICE.G_Now_MS
);

IF fbServiceHeartbeatTimer.Q THEN
    L_Service_Heartbeat_State := NOT L_Service_Heartbeat_State;
END_IF;

GVL_IO.DO_Heartbeat_Pulse := L_Service_Heartbeat_State;
GVL_IO.DO_Active_Status := TRUE;

fbSystemDiagnostics();
PRG_PLC_Arbitration();
PRG_PLC_Fencing_Governor();

GVL_MAIN_PHASE_FEEDBACK.G_Phase_02_Redundancy_Executed := TRUE;
GVL_MAIN_PHASE_FEEDBACK.G_Phase_02_Redundancy_Valid := TRUE;
GVL_MAIN_PHASE_FEEDBACK.G_Phase_02_Redundancy_Status_Text := 'Single active PLC / cold-spare authority phase executed';
GVL_MAIN_PHASE_FEEDBACK.G_Last_Update_MS := GVL_TIME_SERVICE.G_Now_MS;

// >>> BULK_SYNC_ANCHOR: PRG_Main_Phase_02_Redundancy <<<
END_PROGRAM

(* ---- PRG_Main_Phase_03_Input_Safety_Command.st ---- *)
PROGRAM PRG_Main_Phase_03_Input_Safety_Command

GVL_MAIN_PHASE_FEEDBACK.G_Current_Phase := 3;

PRG_IO_Read();
PRG_Input_Quality_Read();
PRG_Input_Processing();

PRG_Heating_Config_Defaults();

PRG_Mode_Manager();
PRG_Presence_Manager();
PRG_Safety_Selector();
PRG_Safety();
PRG_Safety_Operator();
PRG_Safety_Shutdown();
PRG_Safety_Recovery();
PRG_System_Intent();
PRG_Security();
PRG_System_Access_Maintenance();
PRG_User_Adapt_Control();
PRG_Behavior_Adapt_Profile();

PRG_Scenario_Engine();
PRG_System_Scenario_Rules();
PRG_System_Evacuation();
PRG_Policy();
PRG_Heating_Policy_Manager();
PRG_Heating_Policy_Observer();
PRG_System_Coordinator();
PRG_Command_Arbitration();

GVL_MAIN_PHASE_FEEDBACK.G_Phase_03_Input_Safety_Command_Executed := TRUE;
GVL_MAIN_PHASE_FEEDBACK.G_Phase_03_Input_Safety_Command_Valid := TRUE;
GVL_MAIN_PHASE_FEEDBACK.G_Phase_03_Input_Safety_Command_Status_Text := 'Input/safety/command phase executed';
GVL_MAIN_PHASE_FEEDBACK.G_Last_Update_MS := GVL_TIME_SERVICE.G_Now_MS;

// >>> BULK_SYNC_ANCHOR: PRG_Main_Phase_03_Input_Safety_Command <<<
END_PROGRAM

(* ---- PRG_Main_Phase_06_PostOutput_Authority.st ---- *)
PROGRAM PRG_Main_Phase_06_PostOutput_Authority
// MAIN PHASE 12A — post-output authority, physical transaction and causality guards.
// Critical: high. Runs after IO projection to validate authority/physical consistency.

GVL_MAIN_PHASE_FEEDBACK.G_Current_Phase := 6;

PRG_Actuation_Authority_Governor();
PRG_Physical_Transaction_Governor();
PRG_Temporal_Stability_Governor();
PRG_Environmental_Authority_Governor();
PRG_Runtime_Resource_Authority_Governor();
PRG_Semantic_Continuity_Authority_Governor();
PRG_Observability_Truth_Governor();
PRG_Historical_Truth_Governor();
PRG_Global_Authority_Sync_Governor();
PRG_Control_Temporal_Coherence_Governor();
PRG_Actuator_Semantic_Verification_Governor();
PRG_Energy_Causality_Governor();
PRG_Runtime_Sustainability_Governor();

GVL_MAIN_PHASE_FEEDBACK.G_Phase_06_PostOutput_Authority_Executed := TRUE;
GVL_MAIN_PHASE_FEEDBACK.G_Phase_06_PostOutput_Authority_Valid := TRUE;
GVL_MAIN_PHASE_FEEDBACK.G_Phase_06_PostOutput_Authority_Status_Text := 'Post-output authority phase executed';
GVL_MAIN_PHASE_FEEDBACK.G_Last_Update_MS := GVL_TIME_SERVICE.G_Now_MS;

// >>> BULK_SYNC_ANCHOR: PRG_Main_Phase_06_PostOutput_Authority <<<
END_PROGRAM

(* ---- PRG_Modbus_Master.st ---- *)
PROGRAM PRG_Modbus_Master
VAR
    L_i : INT;
    L_Elapsed_MS : UDINT;
END_VAR

// ======================================================
// MODBUS MASTER RUNTIME SCHEDULER
// ======================================================
// Library-independent Modbus master scheduler.
// ======================================================

IF NOT GVL_CONFIG.G_OpenTherm_Enabled THEN

    GVL_MODBUS_MASTER.G_Master_Online := FALSE;
    GVL_MODBUS_MASTER.G_Master_Error := FALSE;

    GVL_MODBUS_MASTER.G_Active := FALSE;
    GVL_MODBUS_MASTER.G_Active_Index := 0;
    GVL_MODBUS_MASTER.G_Active_Sequence := 0;
    GVL_MODBUS_MASTER.G_Active_Start_MS := 0;
    GVL_MODBUS_MASTER.G_Active_Retry_Count := 0;

    FOR L_i := 1 TO 16 DO
        GVL_MODBUS_MASTER.G_Response[L_i].Busy := FALSE;
        GVL_MODBUS_MASTER.G_Response[L_i].Done := FALSE;
        GVL_MODBUS_MASTER.G_Response[L_i].Error := FALSE;
        GVL_MODBUS_MASTER.G_Response[L_i].Error_Code := 0;
    END_FOR;

    RETURN;
END_IF;

GVL_MODBUS_MASTER.G_Master_Online :=
    GVL_MODBUS_RTU_BRIDGE.G_Driver_Online;

GVL_MODBUS_MASTER.G_Master_Error :=
    GVL_MODBUS_RTU_BRIDGE.G_Driver_Error;

// ======================================================
// START NEW TRANSACTION
// ======================================================
IF NOT GVL_MODBUS_MASTER.G_Active THEN

    FOR L_i := 1 TO 16 DO

        IF GVL_MODBUS_MASTER.G_Request[L_i].Enable THEN

            GVL_MODBUS_MASTER.G_Active := TRUE;
            GVL_MODBUS_MASTER.G_Active_Index := L_i;
            GVL_MODBUS_MASTER.G_Active_Sequence :=
                GVL_MODBUS_MASTER.G_Request[L_i].Sequence;

            GVL_MODBUS_MASTER.G_Active_Start_MS :=
                GVL_STATUS.G_System_Time_MS;

            GVL_MODBUS_MASTER.G_Active_Retry_Count := 0;

            GVL_MODBUS_MASTER.G_Response[L_i].Busy := TRUE;
            GVL_MODBUS_MASTER.G_Response[L_i].Done := FALSE;
            GVL_MODBUS_MASTER.G_Response[L_i].Error := FALSE;
            GVL_MODBUS_MASTER.G_Response[L_i].Error_Code := 0;

            EXIT;

        END_IF;

    END_FOR;

END_IF;

// ======================================================
// ACTIVE TRANSACTION SUPERVISION
// ======================================================
IF GVL_MODBUS_MASTER.G_Active THEN

    L_i := GVL_MODBUS_MASTER.G_Active_Index;

    L_Elapsed_MS :=
        GVL_STATUS.G_System_Time_MS -
        GVL_MODBUS_MASTER.G_Active_Start_MS;

    IF GVL_MODBUS_MASTER.G_Response[L_i].Done OR
       GVL_MODBUS_MASTER.G_Response[L_i].Error THEN

        GVL_MODBUS_MASTER.G_Response[L_i].Busy := FALSE;

        GVL_MODBUS_MASTER.G_Active := FALSE;
        GVL_MODBUS_MASTER.G_Last_Transaction_MS :=
            GVL_STATUS.G_System_Time_MS;

        GVL_MODBUS_MASTER.G_Total_Transactions :=
            GVL_MODBUS_MASTER.G_Total_Transactions + 1;

        IF GVL_MODBUS_MASTER.G_Response[L_i].Error THEN
            GVL_MODBUS_MASTER.G_Total_Errors :=
                GVL_MODBUS_MASTER.G_Total_Errors + 1;
        END_IF;

    ELSIF L_Elapsed_MS > GVL_MODBUS_MASTER.G_Request[L_i].Timeout_MS THEN

        GVL_MODBUS_MASTER.G_Active_Retry_Count :=
            GVL_MODBUS_MASTER.G_Active_Retry_Count + 1;

        IF GVL_MODBUS_MASTER.G_Active_Retry_Count >
           GVL_CONFIG.G_Modbus_RTU_Retry_Count THEN

            GVL_MODBUS_MASTER.G_Response[L_i].Busy := FALSE;
            GVL_MODBUS_MASTER.G_Response[L_i].Done := FALSE;
            GVL_MODBUS_MASTER.G_Response[L_i].Error := TRUE;
            GVL_MODBUS_MASTER.G_Response[L_i].Error_Code := 16#0003;

            GVL_MODBUS_MASTER.G_Response[L_i].Last_Sequence :=
                GVL_MODBUS_MASTER.G_Active_Sequence;

            GVL_MODBUS_MASTER.G_Response[L_i].Last_Update_MS :=
                GVL_STATUS.G_System_Time_MS;

            GVL_MODBUS_MASTER.G_Active := FALSE;

            GVL_MODBUS_MASTER.G_Total_Timeouts :=
                GVL_MODBUS_MASTER.G_Total_Timeouts + 1;

            GVL_MODBUS_MASTER.G_Total_Errors :=
                GVL_MODBUS_MASTER.G_Total_Errors + 1;

        ELSE

            GVL_MODBUS_MASTER.G_Active_Start_MS :=
                GVL_STATUS.G_System_Time_MS;

        END_IF;

    END_IF;

END_IF;

END_PROGRAM

(* ---- PRG_Modbus_Register_Scan.st ---- *)
PROGRAM PRG_Modbus_Register_Scan
VAR
    L_Register : UINT;
END_VAR

// ======================================================
// SAFE READ-ONLY MODBUS REGISTER SCAN
// ======================================================
// Safety rules:
//   - FC03/FC04 only.
//   - Never write registers.
//   - Manual enable only.
//   - Limited scan range.
// ======================================================

IF NOT GVL_MODBUS_SCAN.G_Scan_Enable THEN
    GVL_MODBUS_SCAN.G_Scan_Active := FALSE;
    GVL_MODBUS_SCAN.G_Scan_Done := FALSE;
    RETURN;
END_IF;

GVL_MODBUS_SCAN.G_Scan_Active := TRUE;
GVL_MODBUS_SCAN.G_Scan_Error := FALSE;

IF GVL_MODBUS_SCAN.G_Current_Register < GVL_MODBUS_SCAN.G_Start_Register THEN
    GVL_MODBUS_SCAN.G_Current_Register :=
        GVL_MODBUS_SCAN.G_Start_Register;
END_IF;

IF GVL_MODBUS_SCAN.G_Current_Register > GVL_MODBUS_SCAN.G_End_Register THEN
    GVL_MODBUS_SCAN.G_Scan_Active := FALSE;
    GVL_MODBUS_SCAN.G_Scan_Done := TRUE;
    RETURN;
END_IF;

L_Register := GVL_MODBUS_SCAN.G_Current_Register;

// ======================================================
// Issue read-only FC03 request
// ======================================================
GVL_MODBUS_MASTER.G_Request[16].Enable := TRUE;
GVL_MODBUS_MASTER.G_Request[16].Slave_ID := GVL_MODBUS_SCAN.G_Slave_ID;
GVL_MODBUS_MASTER.G_Request[16].Function_Code := MB_FC03_READ_HOLDING_REGISTERS;
GVL_MODBUS_MASTER.G_Request[16].Start_Register := L_Register;
GVL_MODBUS_MASTER.G_Request[16].Register_Count := 1;
GVL_MODBUS_MASTER.G_Request[16].Sequence :=
    GVL_MODBUS_MASTER.G_Request[16].Sequence + 1;
GVL_MODBUS_MASTER.G_Request[16].Timeout_MS := 250;

// ======================================================
// Process response
// ======================================================
IF GVL_MODBUS_MASTER.G_Response[16].Done THEN

    GVL_MODBUS_SCAN.G_Found_Register[L_Register] := TRUE;

    GVL_MODBUS_SCAN.G_Found_Value[L_Register] :=
        GVL_MODBUS_MASTER.G_Response[16].Read_Value[1];

    GVL_MODBUS_SCAN.G_Last_Scan_MS := GVL_STATUS.G_System_Time_MS;

    GVL_MODBUS_SCAN.G_Current_Register :=
        GVL_MODBUS_SCAN.G_Current_Register + 1;

ELSIF GVL_MODBUS_MASTER.G_Response[16].Error THEN

    GVL_MODBUS_SCAN.G_Found_Register[L_Register] := FALSE;

    GVL_MODBUS_SCAN.G_Current_Register :=
        GVL_MODBUS_SCAN.G_Current_Register + 1;

END_IF;

END_PROGRAM

(* ---- PRG_Observability_Authority_Governor.st ---- *)
PROGRAM PRG_Observability_Authority_Governor
VAR
    L_Now_MS : UDINT;
    L_Observability_Valid : BOOL := TRUE;
END_VAR

L_Now_MS := GVL_STATUS.G_System_Time_MS;
L_Observability_Valid := TRUE;

// Fail-safe defaults.
GVL_OBSERVABILITY_AUTHORITY_FABRIC.Observability_Authority_Valid := FALSE;
GVL_OBSERVABILITY_AUTHORITY_FABRIC.Observability_Quarantine_Active := TRUE;
GVL_OBSERVABILITY_AUTHORITY_FABRIC.Observability_Publication_Allowed := FALSE;

GVL_OBSERVABILITY_AUTHORITY_FABRIC.HMI_Authority_Coherent := FALSE;
GVL_OBSERVABILITY_AUTHORITY_FABRIC.Diagnostics_Authority_Coherent := FALSE;
GVL_OBSERVABILITY_AUTHORITY_FABRIC.Blackbox_Authority_Coherent := FALSE;
GVL_OBSERVABILITY_AUTHORITY_FABRIC.Trend_Authority_Coherent := FALSE;
GVL_OBSERVABILITY_AUTHORITY_FABRIC.Alarm_Authority_Coherent := FALSE;

// Revocation blocks authoritative observability.
IF GVL_AUTHORITY_REVOCATION.Authority_Revocation_Active THEN
    L_Observability_Valid := FALSE;
END_IF;

// Restoration must be fully completed.
IF L_Observability_Valid
AND NOT GVL_AUTHORITY_RESTORATION.Authority_Restoration_Completed THEN
    L_Observability_Valid := FALSE;
END_IF;

// Physical authority epoch coherence required.
IF L_Observability_Valid
AND NOT GVL_PHYSICAL_AUTHORITY_EPOCH.Physical_Authority_Epoch_Valid THEN
    L_Observability_Valid := FALSE;
END_IF;

// Authority lineage continuity required.
IF L_Observability_Valid
AND NOT GVL_AUTHORITY_LINEAGE.Authority_Lineage_Valid THEN
    L_Observability_Valid := FALSE;
END_IF;

IF L_Observability_Valid THEN
    GVL_OBSERVABILITY_AUTHORITY_FABRIC.Observability_Authority_Valid := TRUE;
    GVL_OBSERVABILITY_AUTHORITY_FABRIC.Observability_Quarantine_Active := FALSE;
    GVL_OBSERVABILITY_AUTHORITY_FABRIC.Observability_Publication_Allowed := TRUE;

    GVL_OBSERVABILITY_AUTHORITY_FABRIC.HMI_Authority_Coherent := TRUE;
    GVL_OBSERVABILITY_AUTHORITY_FABRIC.Diagnostics_Authority_Coherent := TRUE;
    GVL_OBSERVABILITY_AUTHORITY_FABRIC.Blackbox_Authority_Coherent := TRUE;
    GVL_OBSERVABILITY_AUTHORITY_FABRIC.Trend_Authority_Coherent := TRUE;
    GVL_OBSERVABILITY_AUTHORITY_FABRIC.Alarm_Authority_Coherent := TRUE;

    GVL_OBSERVABILITY_AUTHORITY_FABRIC.Observability_Epoch :=
        GVL_PHYSICAL_AUTHORITY_EPOCH.Physical_Authority_Epoch;

    GVL_OBSERVABILITY_AUTHORITY_FABRIC.Observability_Epoch_Coherent := TRUE;

    GVL_OBSERVABILITY_AUTHORITY_FABRIC.Observability_Last_Update_MS :=
        L_Now_MS;

    GVL_OBSERVABILITY_AUTHORITY_FABRIC.Observability_Lease_Expired := FALSE;
ELSE
    GVL_OBSERVABILITY_AUTHORITY_FABRIC.Observability_Authority_Valid := FALSE;
    GVL_OBSERVABILITY_AUTHORITY_FABRIC.Observability_Quarantine_Active := TRUE;
    GVL_OBSERVABILITY_AUTHORITY_FABRIC.Observability_Publication_Allowed := FALSE;

    GVL_OBSERVABILITY_AUTHORITY_FABRIC.Observability_Lease_Expired := TRUE;

    GVL_OBSERVABILITY_AUTHORITY_FABRIC.Observability_Invalidation_Count :=
        GVL_OBSERVABILITY_AUTHORITY_FABRIC.Observability_Invalidation_Count + 1;
END_IF;

END_PROGRAM

(* ---- PRG_Operational_Intelligence_Governor.st ---- *)
PROGRAM PRG_Operational_Intelligence_Governor
// PASSIVE OPERATIONAL INTELLIGENCE
// NO EXECUTION MUTATION
// NO AUTHORITY MUTATION

GVL_OPERATIONAL_INTELLIGENCE_FABRIC.Operational_Reasoning_Consistency_Valid :=
    GVL_RUNTIME_TRANSITION_SYSTEM.Runtime_Transition_Legal;

GVL_OPERATIONAL_INTELLIGENCE_FABRIC.Runtime_Causal_Projection_Valid :=
    GVL_TEMPORAL_CAUSALITY_CLOSURE_FABRIC.Temporal_Causality_Coherent;

GVL_OPERATIONAL_INTELLIGENCE_FABRIC.Distributed_Operational_Context_Valid :=
    GVL_DISTRIBUTED_SAFETY_REALITY_CONSENSUS_FABRIC.Distributed_Safety_Consensus_Valid;

IF GVL_RUNTIME_TRANSITION_SYSTEM.Illegal_Runtime_Transition_Observed THEN
    GVL_OPERATIONAL_INTELLIGENCE_FABRIC.Active_Degradation_Cause_Available := TRUE;
END_IF;

IF GVL_RUNTIME_TRANSITION_SYSTEM.Recovery_Without_Lineage_Observed THEN
    GVL_OPERATIONAL_INTELLIGENCE_FABRIC.Recovery_Blocker_Observed := TRUE;
END_IF;

END_PROGRAM

(* ---- PRG_Operator_Semantic_Alignment_Governor.st ---- *)
PROGRAM PRG_Operator_Semantic_Alignment_Governor
VAR
    L_Now_MS : UDINT;
    L_Operator_Valid : BOOL := TRUE;
    L_Error_Code : UDINT := 0;
    L_Error_Text : STRING(160) := '';
END_VAR

L_Now_MS := GVL_STATUS.G_System_Time_MS;
L_Operator_Valid := TRUE;
L_Error_Code := 0;
L_Error_Text := '';

// Fail-safe defaults.
GVL_OPERATOR_SEMANTIC_ALIGNMENT.Operator_Semantic_Alignment_Valid := FALSE;
GVL_OPERATOR_SEMANTIC_ALIGNMENT.Operator_Semantic_Alignment_Granted := FALSE;
GVL_OPERATOR_SEMANTIC_ALIGNMENT.Operator_Semantic_Alignment_Quarantine_Active := TRUE;

GVL_OPERATOR_SEMANTIC_ALIGNMENT.HMI_Semantic_State_Coherent := FALSE;
GVL_OPERATOR_SEMANTIC_ALIGNMENT.Operator_Recovery_Intent_Aligned := FALSE;
GVL_OPERATOR_SEMANTIC_ALIGNMENT.Alarm_Semantic_Priority_Coherent := FALSE;
GVL_OPERATOR_SEMANTIC_ALIGNMENT.Runtime_Explanation_Coherent := FALSE;
GVL_OPERATOR_SEMANTIC_ALIGNMENT.Authority_State_Human_Visible := FALSE;

// Semantic preservation required.
IF NOT GVL_SEMANTIC_PRESERVATION_FABRIC.Semantic_Preservation_Granted THEN
    L_Operator_Valid := FALSE;
    L_Error_Code := 40000;
    L_Error_Text := 'Semantic preservation authority not granted';
END_IF;

// Human-machine semantic split-brain detectors.
IF GVL_OPERATOR_SEMANTIC_ALIGNMENT.HMI_Semantic_Lag_Detected THEN
    L_Operator_Valid := FALSE;
    L_Error_Code := 40001;
    L_Error_Text := 'HMI semantic lag detected';
END_IF;

IF GVL_OPERATOR_SEMANTIC_ALIGNMENT.Operator_Interpretation_Skew_Detected THEN
    L_Operator_Valid := FALSE;
    L_Error_Code := 40002;
    L_Error_Text := 'Operator interpretation skew detected';
END_IF;

IF GVL_OPERATOR_SEMANTIC_ALIGNMENT.Alarm_Cognition_Mismatch_Detected THEN
    L_Operator_Valid := FALSE;
    L_Error_Code := 40003;
    L_Error_Text := 'Alarm cognition mismatch detected';
END_IF;

IF GVL_OPERATOR_SEMANTIC_ALIGNMENT.Hidden_Authority_State_Detected THEN
    L_Operator_Valid := FALSE;
    L_Error_Code := 40004;
    L_Error_Text := 'Hidden authority state detected';
END_IF;

IF GVL_OPERATOR_SEMANTIC_ALIGNMENT.Semantic_Explanation_Divergence_Detected THEN
    L_Operator_Valid := FALSE;
    L_Error_Code := 40005;
    L_Error_Text := 'Semantic explanation divergence detected';
END_IF;

IF GVL_OPERATOR_SEMANTIC_ALIGNMENT.Human_Recovery_Misunderstanding_Detected THEN
    L_Operator_Valid := FALSE;
    L_Error_Code := 40006;
    L_Error_Text := 'Human recovery misunderstanding detected';
END_IF;

// Operator cognition coherence validation.
IF L_Operator_Valid
AND NOT GVL_OPERATOR_SEMANTIC_ALIGNMENT.Human_Interpretation_Coherent THEN
    L_Operator_Valid := FALSE;
    L_Error_Code := 40010;
    L_Error_Text := 'Human interpretation coherence invalid';
END_IF;

IF L_Operator_Valid
AND NOT GVL_OPERATOR_SEMANTIC_ALIGNMENT.Adaptive_Runtime_Visibility_Valid THEN
    L_Operator_Valid := FALSE;
    L_Error_Code := 40011;
    L_Error_Text := 'Adaptive runtime visibility invalid';
END_IF;

IF L_Operator_Valid
AND NOT GVL_OPERATOR_SEMANTIC_ALIGNMENT.Semantic_Explanation_Fresh THEN
    L_Operator_Valid := FALSE;
    L_Error_Code := 40012;
    L_Error_Text := 'Semantic explanation freshness invalid';
END_IF;

IF L_Operator_Valid
AND NOT GVL_OPERATOR_SEMANTIC_ALIGNMENT.Operator_Action_Context_Aligned THEN
    L_Operator_Valid := FALSE;
    L_Error_Code := 40013;
    L_Error_Text := 'Operator action context alignment invalid';
END_IF;

IF L_Operator_Valid THEN
    GVL_OPERATOR_SEMANTIC_ALIGNMENT.Operator_Semantic_Alignment_Valid := TRUE;
    GVL_OPERATOR_SEMANTIC_ALIGNMENT.Operator_Semantic_Alignment_Granted := TRUE;
    GVL_OPERATOR_SEMANTIC_ALIGNMENT.Operator_Semantic_Alignment_Quarantine_Active := FALSE;

    GVL_OPERATOR_SEMANTIC_ALIGNMENT.HMI_Semantic_State_Coherent := TRUE;
    GVL_OPERATOR_SEMANTIC_ALIGNMENT.Operator_Recovery_Intent_Aligned := TRUE;
    GVL_OPERATOR_SEMANTIC_ALIGNMENT.Alarm_Semantic_Priority_Coherent := TRUE;
    GVL_OPERATOR_SEMANTIC_ALIGNMENT.Runtime_Explanation_Coherent := TRUE;
    GVL_OPERATOR_SEMANTIC_ALIGNMENT.Authority_State_Human_Visible := TRUE;

    GVL_OPERATOR_SEMANTIC_ALIGNMENT.Operator_Alignment_Epoch :=
        GVL_SEMANTIC_PRESERVATION_FABRIC.Semantic_Preservation_Epoch;

    GVL_OPERATOR_SEMANTIC_ALIGNMENT.Operator_Alignment_Epoch_Coherent := TRUE;

    GVL_OPERATOR_SEMANTIC_ALIGNMENT.Operator_Alignment_Last_Update_MS :=
        L_Now_MS;

    GVL_OPERATOR_SEMANTIC_ALIGNMENT.Operator_Alignment_Lease_Expired := FALSE;

    GVL_OPERATOR_SEMANTIC_ALIGNMENT.Operator_Alignment_Last_Error_Code := 0;
    GVL_OPERATOR_SEMANTIC_ALIGNMENT.Operator_Alignment_Last_Error_Text := '';
ELSE
    GVL_OPERATOR_SEMANTIC_ALIGNMENT.Operator_Semantic_Alignment_Valid := FALSE;
    GVL_OPERATOR_SEMANTIC_ALIGNMENT.Operator_Semantic_Alignment_Granted := FALSE;
    GVL_OPERATOR_SEMANTIC_ALIGNMENT.Operator_Semantic_Alignment_Quarantine_Active := TRUE;

    GVL_OPERATOR_SEMANTIC_ALIGNMENT.Operator_Alignment_Lease_Expired := TRUE;

    GVL_OPERATOR_SEMANTIC_ALIGNMENT.Operator_Alignment_Last_Error_Code :=
        L_Error_Code;

    GVL_OPERATOR_SEMANTIC_ALIGNMENT.Operator_Alignment_Last_Error_Text :=
        L_Error_Text;

    GVL_OPERATOR_SEMANTIC_ALIGNMENT.Operator_Alignment_Invalidation_Count :=
        GVL_OPERATOR_SEMANTIC_ALIGNMENT.Operator_Alignment_Invalidation_Count + 1;
END_IF;

END_PROGRAM

(* ---- PRG_Output_Freshness_Governor.st ---- *)
PROGRAM PRG_Output_Freshness_Governor
VAR
    L_Now_MS : UDINT;
    L_Delta_MS : UDINT;
    L_Output_Valid : BOOL := TRUE;
    L_Error_Code : UDINT := 0;
    L_Error_Text : STRING(160) := '';
END_VAR

L_Now_MS := GVL_STATUS.G_System_Time_MS;
L_Output_Valid := TRUE;
L_Error_Code := 0;
L_Error_Text := '';

IF NOT GVL_RUNTIME_EPOCH.Runtime_Runtime_Barrier_OK THEN
    L_Output_Valid := FALSE;
    L_Error_Code := 6000;
    L_Error_Text := 'Output runtime authority invalid';
END_IF;

IF L_Output_Valid AND (NOT GVL_RUNTIME_EPOCH.Runtime_IO_Publication_Allowed) THEN
    L_Output_Valid := FALSE;
    L_Error_Code := 6001;
    L_Error_Text := 'Output publication not allowed';
END_IF;

IF L_Output_Valid AND (NOT GVL_RUNTIME_SNAPSHOT.Snapshot_Frozen) THEN
    L_Output_Valid := FALSE;
    L_Error_Code := 6100;
    L_Error_Text := 'Runtime snapshot not frozen';
END_IF;

IF L_Output_Valid AND (NOT GVL_RUNTIME_SNAPSHOT.Snapshot_Publication_Allowed) THEN
    L_Output_Valid := FALSE;
    L_Error_Code := 6101;
    L_Error_Text := 'Snapshot publication blocked';
END_IF;

IF L_Output_Valid AND (NOT GVL_RUNTIME_SNAPSHOT.Snapshot_Copy_Valid) THEN
    L_Output_Valid := FALSE;
    L_Error_Code := 6102;
    L_Error_Text := 'Snapshot copy invalid';
END_IF;

IF L_Output_Valid AND (NOT GVL_RUNTIME_SNAPSHOT.Snapshot_Isolation_Valid) THEN
    L_Output_Valid := FALSE;
    L_Error_Code := 6103;
    L_Error_Text := 'Snapshot isolation invalid';
END_IF;

IF L_Output_Valid AND GVL_RUNTIME_SNAPSHOT.Snapshot_Mutation_Detected THEN
    L_Output_Valid := FALSE;
    L_Error_Code := 6104;
    L_Error_Text := 'Snapshot mutation detected';
END_IF;

IF L_Output_Valid AND GVL_DISTRIBUTED_EPOCH.Distributed_Quarantine_Active THEN
    L_Output_Valid := FALSE;
    L_Error_Code := 6200;
    L_Error_Text := 'Distributed reconciliation quarantine active';
END_IF;

IF L_Output_Valid AND (NOT GVL_DISTRIBUTED_SNAPSHOT.Distributed_Publication_Reconciled) THEN
    L_Output_Valid := FALSE;
    L_Error_Code := 6300;
    L_Error_Text := 'Distributed publication reconciliation invalid';
END_IF;

IF L_Output_Valid AND (NOT GVL_DISTRIBUTED_SNAPSHOT.Distributed_Publication_Freeze_Valid) THEN
    L_Output_Valid := FALSE;
    L_Error_Code := 6301;
    L_Error_Text := 'Distributed publication freeze invalid';
END_IF;

IF L_Output_Valid AND (NOT GVL_DISTRIBUTED_SNAPSHOT.Distributed_Snapshot_Consistent) THEN
    L_Output_Valid := FALSE;
    L_Error_Code := 6302;
    L_Error_Text := 'Distributed immutable snapshot inconsistent';
END_IF;

IF L_Output_Valid AND GVL_DISTRIBUTED_SNAPSHOT.Distributed_Snapshot_Quarantine_Active THEN
    L_Output_Valid := FALSE;
    L_Error_Code := 6306;
    L_Error_Text := 'Distributed immutable snapshot quarantine active';
END_IF;

// Finalized distributed publication continuity.
IF L_Output_Valid AND (NOT GVL_DISTRIBUTED_COMMIT.Distributed_Commit_Valid) THEN
    L_Output_Valid := FALSE;
    L_Error_Code := 6400;
    L_Error_Text := 'Distributed commit invalid';
END_IF;

IF L_Output_Valid AND (NOT GVL_DISTRIBUTED_COMMIT.Publication_Prepare_Valid) THEN
    L_Output_Valid := FALSE;
    L_Error_Code := 6402;
    L_Error_Text := 'Distributed publication prepare invalid';
END_IF;

IF L_Output_Valid AND GVL_DISTRIBUTED_COMMIT.Publication_Commit_Requested
   AND (NOT GVL_DISTRIBUTED_COMMIT.Publication_Commit_Confirmed) THEN
    L_Output_Valid := FALSE;
    L_Error_Code := 6403;
    L_Error_Text := 'Distributed publication commit pending';
END_IF;

IF L_Output_Valid AND GVL_DISTRIBUTED_COMMIT.Peer_Commit_Mismatch THEN
    L_Output_Valid := FALSE;
    L_Error_Code := 6404;
    L_Error_Text := 'Distributed peer commit mismatch';
END_IF;

IF L_Output_Valid AND GVL_DISTRIBUTED_COMMIT.Distributed_Commit_Quarantine_Active THEN
    L_Output_Valid := FALSE;
    L_Error_Code := 6401;
    L_Error_Text := 'Distributed commit quarantine active';
END_IF;

IF L_Output_Valid AND GVL_DISTRIBUTED_COMMIT.Commit_Lease_Expired THEN
    L_Output_Valid := FALSE;
    L_Error_Code := 6405;
    L_Error_Text := 'Distributed commit lease expired';
END_IF;

GVL_OUTPUT_EPOCH.Output_Semantic_Continuity_Warning :=
    (NOT GVL_SEMANTIC_PROGRESS.Semantic_Forward_Progress_Valid)
    OR (NOT GVL_SEMANTIC_PROGRESS.Semantic_Execution_Continuity_OK)
    OR GVL_SEMANTIC_PROGRESS.Semantic_Stagnation_Detected
    OR GVL_SEMANTIC_PROGRESS.Semantic_Replay_Suspected
    OR GVL_SEMANTIC_PROGRESS.Semantic_Livelock_Suspected
    OR GVL_SEMANTIC_PROGRESS.Semantic_Deadlock_Suspected
    OR GVL_SEMANTIC_PROGRESS.Semantic_Progress_Lease_Expired
    OR GVL_SEMANTIC_PROGRESS.Semantic_Progress_Quarantine_Active;

// Hard semantic continuity invalidation.
IF L_Output_Valid
AND GVL_OUTPUT_EPOCH.Output_Semantic_Continuity_Warning
THEN
    L_Output_Valid := FALSE;
    L_Error_Code := 6500;
    L_Error_Text := 'Semantic continuity invalid';
END_IF;

IF L_Output_Valid THEN
    IF GVL_OUTPUT_EPOCH.Output_Runtime_Epoch > GVL_RUNTIME_EPOCH.Runtime_Epoch THEN
        L_Output_Valid := FALSE;
        L_Error_Code := 6002;
        L_Error_Text := 'Output epoch ahead of runtime epoch';
    END_IF;
END_IF;

L_Delta_MS := L_Now_MS - GVL_OUTPUT_EPOCH.Output_Last_Refresh_MS;

IF L_Output_Valid AND GVL_OUTPUT_EPOCH.Output_Lease_Active THEN
    IF L_Delta_MS > GVL_OUTPUT_EPOCH.Output_Lease_Timeout_MS THEN
        L_Output_Valid := FALSE;
        L_Error_Code := 6003;
        L_Error_Text := 'Output lease expired';
    END_IF;
END_IF;

IF L_Output_Valid THEN
    GVL_OUTPUT_EPOCH.Output_Publication_Epoch := GVL_OUTPUT_EPOCH.Output_Publication_Epoch + 1;

    GVL_OUTPUT_EPOCH.Output_Publication_Valid := TRUE;
    GVL_OUTPUT_EPOCH.Output_Lease_Active := TRUE;
    GVL_OUTPUT_EPOCH.Output_Lease_Expired := FALSE;

    GVL_OUTPUT_EPOCH.Output_Runtime_Epoch := GVL_RUNTIME_EPOCH.Runtime_Epoch;
    GVL_OUTPUT_EPOCH.Output_Runtime_Epoch_Valid := TRUE;

    GVL_OUTPUT_EPOCH.Output_Last_Publication_MS := L_Now_MS;
    GVL_OUTPUT_EPOCH.Output_Last_Refresh_MS := L_Now_MS;

    IF GVL_CONVERGENCE.Convergence_Release_Allowed THEN
        GVL_OUTPUT_EPOCH.Output_Stale_Detected := FALSE;
        GVL_OUTPUT_EPOCH.Output_Forced_Safe_Decay := FALSE;
    END_IF;

    GVL_OUTPUT_EPOCH.Output_Last_Error_Code := 0;
    GVL_OUTPUT_EPOCH.Output_Last_Error_Text := '';
ELSE
    GVL_OUTPUT_EPOCH.Output_Publication_Valid := FALSE;
    GVL_OUTPUT_EPOCH.Output_Lease_Expired := TRUE;
    GVL_OUTPUT_EPOCH.Output_Stale_Detected := TRUE;
    GVL_OUTPUT_EPOCH.Output_Forced_Safe_Decay := TRUE;

    GVL_OUTPUT_EPOCH.Output_Last_Invalidation_MS := L_Now_MS;
    GVL_OUTPUT_EPOCH.Output_Last_Error_Code := L_Error_Code;
    GVL_OUTPUT_EPOCH.Output_Last_Error_Text := L_Error_Text;
END_IF;
END_PROGRAM

(* ---- PRG_Physical_Authority_Epoch_Governor.st ---- *)
PROGRAM PRG_Physical_Authority_Epoch_Governor
VAR
    L_Now_MS : UDINT;
    L_Epoch_Valid : BOOL := TRUE;
    L_Error_Code : UDINT := 0;
    L_Error_Text : STRING(160) := '';
    L_Global_Epoch : UDINT;
END_VAR

L_Now_MS := GVL_STATUS.G_System_Time_MS;
L_Epoch_Valid := TRUE;
L_Error_Code := 0;
L_Error_Text := '';

// Fail-safe defaults.
GVL_PHYSICAL_AUTHORITY_EPOCH.Physical_Authority_Epoch_Valid := FALSE;
GVL_PHYSICAL_AUTHORITY_EPOCH.Snapshot_Epoch_Coherent := FALSE;
GVL_PHYSICAL_AUTHORITY_EPOCH.Consensus_Epoch_Coherent := FALSE;
GVL_PHYSICAL_AUTHORITY_EPOCH.Causality_Epoch_Coherent := FALSE;
GVL_PHYSICAL_AUTHORITY_EPOCH.PreOutput_Epoch_Coherent := FALSE;

L_Global_Epoch := GVL_PHYSICAL_SNAPSHOT.Physical_Snapshot_Epoch;

// Snapshot epoch is the authoritative physical world epoch.
IF GVL_PHYSICAL_SNAPSHOT.Physical_Snapshot_Epoch = 0 THEN
    L_Epoch_Valid := FALSE;
    L_Error_Code := 24000;
    L_Error_Text := 'Physical snapshot epoch invalid';
END_IF;

// Consensus must validate the same immutable world.
IF L_Epoch_Valid
AND (GVL_SENSOR_CONSENSUS.Sensor_Consensus_Epoch <> L_Global_Epoch) THEN
    GVL_PHYSICAL_AUTHORITY_EPOCH.Cross_Cycle_Epoch_Skew_Detected := TRUE;

    L_Epoch_Valid := FALSE;
    L_Error_Code := 24001;
    L_Error_Text := 'Sensor consensus epoch skew detected';
END_IF;

// Telemetry causality must validate the same immutable world.
IF L_Epoch_Valid
AND (GVL_TELEMETRY.Telemetry_Epoch <> L_Global_Epoch) THEN
    GVL_PHYSICAL_AUTHORITY_EPOCH.Cross_Cycle_Epoch_Skew_Detected := TRUE;

    L_Epoch_Valid := FALSE;
    L_Error_Code := 24002;
    L_Error_Text := 'Telemetry epoch skew detected';
END_IF;

// Output publication epoch must remain coherent.
IF L_Epoch_Valid
AND (GVL_OUTPUT_EPOCH.Output_Publication_Epoch <> L_Global_Epoch) THEN
    GVL_PHYSICAL_AUTHORITY_EPOCH.Partial_Epoch_Advancement_Detected := TRUE;

    L_Epoch_Valid := FALSE;
    L_Error_Code := 24003;
    L_Error_Text := 'Output publication epoch skew detected';
END_IF;

IF L_Epoch_Valid
AND GVL_PHYSICAL_AUTHORITY_EPOCH.Physical_Epoch_Replay_Suspected THEN
    L_Epoch_Valid := FALSE;
    L_Error_Code := 24004;
    L_Error_Text := 'Physical authority epoch replay suspected';
END_IF;

IF L_Epoch_Valid
AND GVL_PHYSICAL_AUTHORITY_EPOCH.Physical_Epoch_Drift_Detected THEN
    L_Epoch_Valid := FALSE;
    L_Error_Code := 24005;
    L_Error_Text := 'Physical authority epoch drift detected';
END_IF;

IF L_Epoch_Valid THEN
    GVL_PHYSICAL_AUTHORITY_EPOCH.Physical_Authority_Epoch := L_Global_Epoch;
    GVL_PHYSICAL_AUTHORITY_EPOCH.Physical_Authority_Epoch_Valid := TRUE;

    GVL_PHYSICAL_AUTHORITY_EPOCH.Snapshot_Epoch_Coherent := TRUE;
    GVL_PHYSICAL_AUTHORITY_EPOCH.Consensus_Epoch_Coherent := TRUE;
    GVL_PHYSICAL_AUTHORITY_EPOCH.Causality_Epoch_Coherent := TRUE;
    GVL_PHYSICAL_AUTHORITY_EPOCH.PreOutput_Epoch_Coherent := TRUE;

    GVL_PHYSICAL_AUTHORITY_EPOCH.Physical_Authority_Lease_Expired := FALSE;
    GVL_PHYSICAL_AUTHORITY_EPOCH.Physical_Authority_Quarantine_Active := FALSE;

    GVL_PHYSICAL_AUTHORITY_EPOCH.Physical_Authority_Last_Update_MS := L_Now_MS;

    GVL_PHYSICAL_AUTHORITY_EPOCH.Physical_Authority_Last_Error_Code := 0;
    GVL_PHYSICAL_AUTHORITY_EPOCH.Physical_Authority_Last_Error_Text := '';
ELSE
    GVL_PHYSICAL_AUTHORITY_EPOCH.Physical_Authority_Epoch_Valid := FALSE;

    GVL_PHYSICAL_AUTHORITY_EPOCH.Physical_Authority_Lease_Expired := TRUE;
    GVL_PHYSICAL_AUTHORITY_EPOCH.Physical_Authority_Quarantine_Active := TRUE;

    GVL_PHYSICAL_AUTHORITY_EPOCH.Physical_Authority_Last_Error_Code := L_Error_Code;
    GVL_PHYSICAL_AUTHORITY_EPOCH.Physical_Authority_Last_Error_Text := L_Error_Text;

    GVL_PHYSICAL_AUTHORITY_EPOCH.Physical_Authority_Invalidation_Count :=
        GVL_PHYSICAL_AUTHORITY_EPOCH.Physical_Authority_Invalidation_Count + 1;
END_IF;

END_PROGRAM

(* ---- PRG_Physical_Safety_Projection_Governor.st ---- *)
PROGRAM PRG_Physical_Safety_Projection_Governor
IF GVL_SAFETY_OBSERVABILITY_TRUTH_FABRIC.Safety_Observability_Truth_Granted
AND NOT GVL_PHYSICAL_SAFETY_PROJECTION_FABRIC.Physical_Safety_Projection_Drift_Detected
AND NOT GVL_PHYSICAL_SAFETY_PROJECTION_FABRIC.Hidden_Unsafe_Physical_State_Detected
AND NOT GVL_PHYSICAL_SAFETY_PROJECTION_FABRIC.Unsafe_Projection_Backfill_Detected THEN

    GVL_PHYSICAL_SAFETY_PROJECTION_FABRIC.Physical_Safety_Projection_Valid := TRUE;
    GVL_PHYSICAL_SAFETY_PROJECTION_FABRIC.Physical_Safety_Projection_Granted := TRUE;
    GVL_PHYSICAL_SAFETY_PROJECTION_FABRIC.Physical_Plant_Safety_Projection_Stable := TRUE;
    GVL_PHYSICAL_SAFETY_PROJECTION_FABRIC.Energy_State_Safety_Projection_Valid := TRUE;
    GVL_PHYSICAL_SAFETY_PROJECTION_FABRIC.Recovery_State_Safety_Projection_Valid := TRUE;
END_IF;
END_PROGRAM

(* ---- PRG_PLC_A.st ---- *)
PROGRAM PRG_PLC_A
VAR
    // Специфичная логика для ПЛК А
END_VAR

// Вызов основной программы
PRG_System();
// >>> BULK_SYNC_ANCHOR: PRG_PLC_A <<<
END_PROGRAM
